	//nInputStatus
	ingPressureControl 		: BOOL;
	ingPositionControl 		: BOOL;
	isValveOpen 			: BOOL;
	isValveNotInitialized 	: BOOL;	
	isValveClosed 			: BOOL;
	isValveFaultState 		: BOOL;
	ingValveInitializing 	: BOOL;
	ingHoldState 			: BOOL;
	isPressureControl:BOOL;
	
	// Vacuum Pump Status
	isPumpFault				: BOOL;
	isPumpWarning			: BOOL;
	isPumpAlarm				: BOOL;
	isFBRunning				: BOOL;
 	isPumpRunning			: BOOL;
	//wSetPoint 			: WORD; //Set Point
	nTValveMode 		: USINT := 0; //Valve Mode
	bPumpOn				: BOOL;
	bPumpReset			: BOOL;	//Input from IQ-PLUS Throttle Valve
	
	wTypedControlValue 	: WORD;
	wOutputSVBytes : outWord; //Word to Byte variable
	nSetType 			: USINT; //1:Pressure Conrol, 2:Position Control
	
	wByteCDG1_PV 			: WORD; //CDG1 Current Pressure, Not Used
	wByteCDG2_PV 			: WORD; //CDG2 Current Pressure
	wByteValvePosition_PV : WORD; //Current Valve Position (0~100%)
	nInputStatusOld : USINT := 9; //Value Change Monitoring, First Temp value
	wByteValvePosition_PV_Monitoring: WORD;
	CDG1_RealValue: REAL;
	nOutputSetType:USINT; //1:Pressure Conrol, 2:Position Control
	CDG_1_Value_RealType: REAL;
END_VAR

VAR CONSTANT
	//Conversion Parameter
	SetPointFactor : REAL := 327.67; //Range 0~7FFFh
	PressureFactor : REAL := 24.576;	//Range 0~6000h
END_VAR

//jhkang_251112
////Model : IQ Plus 
////Pressure Range : 0 ~ 1,000 Torr
//IF GVL_COMMAND_FROM_UI.CMD_THROTTLE_PRESSURE_POSITION_MODE THEN //true: Pressure False:Position
//	GVL_DEVICE_NET_IQ_PLUS.nOutputSetType := 1; // Pressure Control
//ELSE
//	GVL_DEVICE_NET_IQ_PLUS.nOutputSetType := 2; // Position Control
//END_IF

//nSetType := GVL_DEVICE_NET_IQ_PLUS.nOutputSetType;
//nOutputSetType:=nSetType;


//_DIgitalInput();
//_CalData();
//_DigitalOutput();


//nTValveMode := WORD_TO_USINT(GVL_IO.aOutputCmd[2]); //Throttle Valve Mode Setting 0:Normal 1:Close 2:Open 3:Hold 4:Reset

ACTION _CalData:
//jhkang_251112
//// nOutputMode
//// 0 : uses setpoint and setpoint type to control the valve.
//// 1 : Does not use setpoint and setpoint type to operate the valve.
//// 2 : Does not use setpoint and setpoint type to operate the valve.
//// 3 : Holds valve in current position.
//// 4 : Reset the controller.

//GVL_IO.nIQPLUS_SetType 	:= GVL_DEVICE_NET_IQ_PLUS.nOutputSetType;
//GVL_IO.nIQPLUS_Mode 	:= GVL_DEVICE_NET_IQ_PLUS.nOutputMode;
//GVL_DEVICE_NET_IQ_PLUS.nOutputMode := GVL_COMMAND_FROM_UI.CMD_THROTTLE_OUTPUT_MODE;
//GVL_INTERFACE_UI.aMonitoring_PV[E_Morning_Index.E_Morning_TV_Position] := wByteValvePosition_PV/SetPointFactor;

//(* Read from Device Value *)
//// 2USINT to WORD
//wByteCDG1_PV 		:= USINT_TO_WORD_jh(GVL_DEVICE_NET_IQ_PLUS.aInputPressurePV_CDG1);
//wByteCDG2_PV 		:= USINT_TO_WORD_jh(GVL_DEVICE_NET_IQ_PLUS.aInputPressurePV_CDG2);
//wByteValvePosition_PV:= USINT_TO_WORD_jh(GVL_DEVICE_NET_IQ_PLUS.aInputValvePosionPV);
//wByteValvePosition_PV_Monitoring:=REAL_TO_WORD(wByteValvePosition_PV/SetPointFactor);
//GVL_INTERFACE_UI.aMonitoring_PV[12] := wByteValvePosition_PV_Monitoring;




//wControlValue		:= GVL_IO.wIqPlus_CV;

////From IQ Plus
//CDG1_RealValue :=wByteCDG1_PV/PressureFactor; 
//GVL_IO.wIqPlus_CDG1_PV 	:= REAL_TO_WORD(wByteCDG1_PV/PressureFactor);
//GVL_IO.wIqPlus_CDG2_PV:=GVL_IO.wIqPlus_CDG1_PV;

//IF GVL_IO.wIqPlus_CDG1_PV > 1000 OR GVL_IO.wIqPlus_CDG1_PV <=5 THEN
//	GVL_IO.wIqPlus_CDG1_PV:=0;
//	GVL_IO.wIqPlus_CDG2_PV:=0;
//END_IF

//CDG_1_Value_RealType:=wByteCDG1_PV/PressureFactor;


////nSetType //1:Pressure Conrol, 2:Position Control

//IF GVL_DEVICE_NET_IQ_PLUS.nOutputMode = 0 AND nSetType = 1 THEN(*Pressure Mode*)
//	wTypedControlValue := REAL_TO_WORD(wControlValue * SetPointFactor * 0.1); //Pressure Control
//ELSIF GVL_DEVICE_NET_IQ_PLUS.nOutputMode = 0 AND nSetType = 2 THEN (*Position Mode*)
//	wTypedControlValue := REAL_TO_WORD(wControlValue * SetPointFactor); // Position Control
//END_IF

//wOutputSVBytes 		:= WORD_TO_USINT_Bit(wTypedControlValue);
//GVL_DEVICE_NET_IQ_PLUS.aOutputSVBytes[1] 	:= wOutputSVBytes.Lower;
//GVL_DEVICE_NET_IQ_PLUS.aOutputSVBytes[2] 	:= wOutputSVBytes.Upper;

////Valve Status Initailize
//IF GVL_DEVICE_NET_IQ_PLUS.nInputStatus <> nInputStatusOld THEN
//	// Staus Initializing
//	ingPressureControl := FALSE;
//	ingPositionControl := FALSE;
//	isValveOpen := FALSE;
//	isValveNotInitialized := FALSE;	
//	isValveClosed := FALSE;
//	isValveFaultState := FALSE;
//	ingValveInitializing := FALSE;
//	ingHoldState := FALSE;
//	isPressureControl:=FALSE;
//	// Status Update	
//	nInputStatusOld := GVL_DEVICE_NET_IQ_PLUS.nInputStatus;
//END_IF



////Update Valve Status
//CASE GVL_DEVICE_NET_IQ_PLUS.nInputStatus OF
//	0 : ingPressureControl := TRUE; //Pressure Control Performing.
//	1 : ingPositionControl := TRUE; //Position Control Performing.	
//	2 : isValveOpen := TRUE; //Valve Open, Stopped, Not Controlling.
//	3 : isValveNotInitialized := TRUE; //Valve not initialized power on or RESET Command.
//	4 : isValveClosed := TRUE; //Valve Closed, Stopped, Not Controlling.
//	5 : isValveFaultState := TRUE; //Has faulted during valve initialization or operation.
//	6 : ingValveInitializing := TRUE; //Initailizing Process.
//	7 :	isPressureControl:=TRUE;
//	8 : ingHoldState := TRUE; //intermediate position, not at open or close and not controlling pressure.
//END_CASE
END_ACTION

ACTION _DigitalInput:

//jhkang_251112
//(* Command *)

//bPumpOn:= GVL_COMMAND_FROM_UI.CMD_VACUUM_PUMP_ON;
//bPumpReset:=GVL_COMMAND_FROM_UI.CMD_VACUUM_PUMP_RESET;
//(* Read from Power Distribution Pannel *)
//bVacuumPumpCB		:= GVL_IO_GAS_CABINET.DI_02_VacuumPumpELCB;
//bThrottleValveCP 	:= GVL_IO_GAS_CABINET.DI_02_T_VCP;

//(* Read from Vacuum Pump *)
//isPumpFault			:= GVL_IO_REACTOR_CABINET.DI_02_VacuumPumpFail;
//isPumpWarning		:= GVL_IO_REACTOR_CABINET.DI_02_VacuumPumpWarning;
//isPumpAlarm			:= GVL_IO_REACTOR_CABINET.DI_02_VacuumPumpAlarm;
//isPumpRunning		:= GVL_IO_REACTOR_CABINET.DI_02_VacuumPumpFBRunning;
//isFBRunning			:= GVL_IO_REACTOR_CABINET.DI_02_VacuumPumpRunning;


//GVL_IO.isPumpRunning := GVL_IO_REACTOR_CABINET.DI_02_VacuumPumpFBRunning;
END_ACTION

ACTION _DigitalOutput:
//GVL_IO.aDigitalOutputIO[2].2 := bPumpOn; //Pump On
//GVL_IO.aDigitalOutputIO[2].3 := bPumpReset; // Pump Reset

GVL_IO_REACTOR_CABINET.DO_05_VacuumPumpStart_Stop := bPumpOn;
GVL_IO_REACTOR_CABINET.DO_05_VacuumPumpReset := bPumpReset;
END_ACTION

END_PROGRAM

// ---- POUs/P13_LineHeater.TcPOU
PROGRAM P13_LineHeater
VAR
	rTemperatureSV 		: ARRAY[1..8]OF REAL;
	bAutoTuneSV 		: ARRAY[1..8]OF BOOL;

	rTemperaturePV 		: ARRAY[1..8]OF REAL;
	isLineHeater_Run	: ARRAY[1..8]OF BOOL;
	isLineHeater_ATune	: ARRAY[1..8]OF BOOL;
	isLineHeater_Err	: ARRAY[1..8]OF BOOL;

	TimeOnDelay			: TON; //Time delay after Power ON of Thermal Bath
	TimeCycle			: TON;
	nComMode 			: INT; // //1 = PV Req, 2 = STATUS Req, 3 = SV Write, 4 = AutoTune On/Off
	nCount 				: INT;
	rTemperatureTV 		: ARRAY[1..8]OF REAL;
	bAutoTuneTV			: ARRAY[1..8]OF BOOL;

	//for sending variable
	TimeWaitSend		:TON;
	bSendingEnable 		: BOOL:=TRUE; // Check the Sending Stage
	bSetValueMode 		: BOOL;
	fbSend				: SendString;
	sSendString 		: STRING;
	bSendBusy			: BOOL;
	bSendingOK 			: BOOL; //v1
	eSendErrorID		: ComError_t;
	
	// for received variable
	TimeWaitReceive		:TON;
	fbReceive			: ReceiveString;
	sReceivedString		: STRING;
	bStringReceived		: BOOL;
	bReceiveBusy		: BOOL;
	bReceiveError		: BOOL;
	eReceiveErrorID		: ComError_t;
	bReceiveTimeout		: BOOL;
	bReceivedOK 		: BOOL;
	hStrReceivedST		: STRING;
	hStrReceivedPV		: STRING;
	
	nHeaterNumber 		: INT := 1;
	sHeaterNumber 		: STRING := '1';
	sReceivedHeaterNumber : STRING;
	nReceivedHeaterNumber : INT;
	sReceivedAffirmation : STRING;
	sReceivedData 		: STRING;
	nHeaterStrPositionPV : INT:= 11; //Received String Start Position
	nDecimal			:INT;
	nSendStrCounter		:INT := 1;
	bReset : BOOL;
	sTest : STRING;
	nStrPosition : INT;
	nHeaterNumberPV : INT;
	sTemperaturePV : STRING;
	(* Input *)
	bLineHeaterCB		: BOOL;
	bLineHeaterCP		: BYTE;
END_VAR

_DIgitalInput();
TimeOnDelay(IN:= GVL_IO_GAS_CABINET.DI_02_LineHeatersELCB, PT :=T#5S); //Time Delay after a Thermal Bath MC ON

IF TimeOnDelay.Q THEN
	
	_GetSP();
	
	TimeOnDelay(IN:=FALSE);
	FOR nHeaterNumber:= 1 TO 8 DO
		IF (rTemperatureTV[nHeaterNumber] <> rTemperatureSV[nHeaterNumber]) THEN
			rTemperatureTV[nHeaterNumber] := rTemperatureSV[nHeaterNumber];
			
			_SendTemp();
		END_IF
	END_FOR
END_IF


_Update_Data();

ACTION _DigitalInput:
bLineHeaterCB	:= GVL_IO_GAS_CABINET.DI_02_LineHeatersELCB;

bLineHeaterCP.0 	:= GVL_IO_GAS_CABINET.DI_03_LineHeater_1CP;
bLineHeaterCP.1 	:= GVL_IO_GAS_CABINET.DI_03_LineHeater_2CP;
bLineHeaterCP.2 	:= GVL_IO_GAS_CABINET.DI_03_LineHeater_3CP;
bLineHeaterCP.3 	:= GVL_IO_GAS_CABINET.DI_03_LineHeater_4CP;
bLineHeaterCP.4 	:= GVL_IO_GAS_CABINET.DI_03_LineHeater_5CP;
bLineHeaterCP.5 	:= GVL_IO_GAS_CABINET.DI_04_LineHeater_6CP;
bLineHeaterCP.6 	:= GVL_IO_GAS_CABINET.DI_04_LineHeater_7CP;
bLineHeaterCP.7 	:= GVL_IO_GAS_CABINET.DI_04_LineHeater_8CP;
END_ACTION

ACTION _GetSP:
//jhkang_251112
//rTemperatureSV[1] := GVL_IO.aInterlockSet[13];
//rTemperatureSV[2] := GVL_IO.aInterlockSet[14];
//rTemperatureSV[3] := GVL_IO.aInterlockSet[15];
//rTemperatureSV[4] := GVL_IO.aInterlockSet[16];
//rTemperatureSV[5] := GVL_IO.aInterlockSet[17];
//rTemperatureSV[6] := GVL_IO.aInterlockSet[18];
//rTemperatureSV[7] := GVL_IO.aInterlockSet[19];
//rTemperatureSV[8] := GVL_IO.aInterlockSet[20];
END_ACTION

ACTION _SendTemp:
CASE nHeaterNumber OF
	1:
		GVL.fbLineHeater_Manager._SendModbusCommand(sendMessage:=F_Temp_Write_Set_Point(Module_Number:=1,CommandIndex:=16#0
																,Write_Value:=REAL_TO_WORD(rTemperatureSV[nHeaterNumber])));
	2:
		GVL.fbLineHeater_Manager._SendModbusCommand(sendMessage:=F_Temp_Write_Set_Point(Module_Number:=1,CommandIndex:=16#03E8
																,Write_Value:=REAL_TO_WORD(rTemperatureSV[nHeaterNumber])));
	3:
		GVL.fbLineHeater_Manager._SendModbusCommand(sendMessage:=F_Temp_Write_Set_Point(Module_Number:=1,CommandIndex:=16#07D0
																,Write_Value:=REAL_TO_WORD(rTemperatureSV[nHeaterNumber])));
	4:
		GVL.fbLineHeater_Manager._SendModbusCommand(sendMessage:=F_Temp_Write_Set_Point(Module_Number:=1,CommandIndex:=16#0BB8
																,Write_Value:=REAL_TO_WORD(rTemperatureSV[nHeaterNumber])));
																
	(*Change Module Number*)															
	5:
		GVL.fbLineHeater_Manager._SendModbusCommand(sendMessage:=F_Temp_Write_Set_Point(Module_Number:=2,CommandIndex:=16#0
																,Write_Value:=REAL_TO_WORD(rTemperatureSV[nHeaterNumber])));
	6:
		GVL.fbLineHeater_Manager._SendModbusCommand(sendMessage:=F_Temp_Write_Set_Point(Module_Number:=2,CommandIndex:=16#03E8
																,Write_Value:=REAL_TO_WORD(rTemperatureSV[nHeaterNumber])));
	7:
		GVL.fbLineHeater_Manager._SendModbusCommand(sendMessage:=F_Temp_Write_Set_Point(Module_Number:=2,CommandIndex:=16#07D0
																,Write_Value:=REAL_TO_WORD(rTemperatureSV[nHeaterNumber])));
	8:
		GVL.fbLineHeater_Manager._SendModbusCommand(sendMessage:=F_Temp_Write_Set_Point(Module_Number:=2,CommandIndex:=16#0BB8
																,Write_Value:=REAL_TO_WORD(rTemperatureSV[nHeaterNumber])));
END_CASE
END_ACTION

ACTION _Update_Data:
//jhkang_251112

//rTemperaturePV[1] := GVL_Serial.LineHeater_data_1.LINE_HEATER_CH_1_PV_VALUE;
//rTemperaturePV[2] := GVL_Serial.LineHeater_data_1.LINE_HEATER_CH_2_PV_VALUE;
//rTemperaturePV[3] := GVL_Serial.LineHeater_data_1.LINE_HEATER_CH_3_PV_VALUE;
//rTemperaturePV[4] := GVL_Serial.LineHeater_data_1.LINE_HEATER_CH_4_PV_VALUE;

//rTemperaturePV[5] := GVL_Serial.LineHeater_data_2.LINE_HEATER_CH_1_PV_VALUE;
//rTemperaturePV[6] := GVL_Serial.LineHeater_data_2.LINE_HEATER_CH_2_PV_VALUE;
//rTemperaturePV[7] := GVL_Serial.LineHeater_data_2.LINE_HEATER_CH_3_PV_VALUE;
//rTemperaturePV[8] := GVL_Serial.LineHeater_data_2.LINE_HEATER_CH_4_PV_VALUE;

//GVL_IO.aLineHeater_rTemperaturePV := rTemperaturePV;
END_ACTION

END_PROGRAM

// ---- POUs/P14_ThermalBath.TcPOU
PROGRAM P14_ThermalBath
VAR
	rTemperatureSV 		: ARRAY[1..6]OF REAL;

	(* Input from Device *)
	bTempDeviationAlarm	: ARRAY[1..6] OF BOOL;
	bCutOffAlarm		: ARRAY[1..6] OF BOOL;
	
	rTemperature_PV 		: ARRAY[1..6]OF REAL;
	isBath_Err 			: ARRAY[1..6]OF BOOL;
	isBath_TC_Broken 	: ARRAY[1..6]OF BOOL ; 

	//for send variable
	TimeOnDelay	: TON; //Time delay after Power ON of Thermal Bath
	TimeCycle			: TON;
	TimeWaitSend		: TON;
	TimeWaitReceive		: TON;
	bSendingEnable 		: BOOL:=TRUE; // Check the Sending Stage
	bSetValueMode 		: BOOL;
	rTemperatureTV 		: ARRAY[1..6]OF REAL;
	fbSend				: SendString;
	sSendString 		: STRING;
	bSendBusy			: BOOL;
	bSendingOK 			: BOOL;
	eSendErrorID		: ComError_t;

	// for received variable
	fbReceive			: ReceiveString;
	sReceivedString		: STRING;
	bStringReceived		: BOOL;
	bReceiveBusy		: BOOL;
	bReceiveError		: BOOL;
	eReceiveErrorID		: ComError_t;
	bReceiveTimeout		: BOOL;
	bReceivedOK 		: BOOL;
	
	nBathNumber 		: INT := 1;
	sBathNumber 		: STRING := '1';
	sReceivedBathNumber : STRING;
	nReceivedBathNumber : INT;
	sReceivedAffirmation : STRING;
	sReceivedData 		: STRING;
	
	(* Input *)
	bThermalBathCB		: BOOL;
	TonSendTmeOut: TON;
	SendTimeOutCount: DINT;
END_VAR


(* Read from Power Distribution Pannel *)
_DigitalInput();

// make a sending string
TimeCycle(IN := TimeOnDelay.Q, PT := T#1000MS); //Cycle for Serial Communication
IF TimeCycle.Q = TRUE THEN
	TimeCycle(IN := FALSE);
	_01_SendMessage();
END_IF

_02_ReceivedMessage();


TonSendTmeOut(IN:=bSendingEnable = FALSE ,PT:=T#10S);
IF TonSendTmeOut.Q THEN
	SendTimeOutCount := SendTimeOutCount+1;
	
	TonSendTmeOut(IN:=false);
	bSendingEnable:=TRUE;
END_IF

ACTION _01_SendMessage:

// Make a sending string Set value or Request value 
IF bSendingEnable = TRUE THEN
	
	nBathNumber := nBathNumber + 1;
	IF nBathNumber > 4 THEN
		nBathNumber := 1;
	END_IF
	
	bSendingEnable := FALSE;
	bReceivedOK := FALSE;
	bSetValueMode := FALSE;
	
	//Target value(Bath) Set value
	IF (rTemperatureTV[nBathNumber] <> rTemperatureSV[nBathNumber])  THEN
		rTemperatureTV[nBathNumber] := rTemperatureSV[nBathNumber];
		sSendString := Real_To_String_ThermalBath(rTemperatureTV[nBathNumber],nBathNumber); //Send a SetValue=10.0 '$0201WSV100100$03'
		bSetValueMode := TRUE;
	ELSE
		sBathNumber := INT_TO_STRING(nBathNumber);
		sSendString := INSERT('$020RPV1$03',sBathNumber,2); //Request a PV
		bSetValueMode := FALSE;
	END_IF
	
	// Send string	
	fbSend(	SendString:= sSendString,
		TXbuffer:= GVL_Serial.TxBufferTB,
		Busy=> bSendBusy,
		Error=> );
		
	IF fbSend.Error <> COMERROR_NOERROR THEN
		eSendErrorID := fbSend.Error;
		bSendingOK := FALSE;
	ELSE
		eSendErrorID := COMERROR_NOERROR;
		bSendingOK := TRUE;
	END_IF
END_IF
END_ACTION

ACTION _02_ReceivedMessage:
//	Receive string data:
//	The block receives any data strings beginning with a STX ($02) and ending with an ETX ($03) character.
TimeWaitReceive(IN := bSendingOK, PT := T#250MS); //Wait receiving data
IF TimeWaitReceive.Q THEN
	TimeWaitReceive(IN:= FALSE);
	fbReceive(
		Prefix:= '$02',
		Suffix:= '$03',
		Timeout:= T#1S,
		ReceivedString:= sReceivedString,
		RXbuffer:= GVL_Serial.RxBufferTB,
		StringReceived=> bStringReceived,
		Busy=> bReceiveBusy,
		Error=> ,
		RxTimeout=> bReceiveTimeout );
		
	IF bReceiveTimeout THEN
		isBath_Err[nReceivedBathNumber] := TRUE;
		bReceiveTimeout := FALSE;
	END_IF
	
	IF fbReceive.Error <> COMERROR_NOERROR THEN
		eReceiveErrorID := fbReceive.Error;
	END_IF
	
	IF bStringReceived THEN
		bStringReceived :=FALSE;
		bReceivedOK := TRUE;
		bSendingEnable := TRUE;
		sReceivedBathNumber := MID(STR:=sReceivedString, len:=1, pos:=3); //ReceivedString : '$0201$06PV100250$03'
		nReceivedBathNumber := STRING_TO_INT(sReceivedBathNumber);
		sReceivedAffirmation := MID(STR:=sReceivedString, len:=1, pos:=4); //Affirmation
		
		IF bSetValueMode THEN //Write SV Mode
			IF sReceivedAffirmation = '$06' THEN //'$06' ReceivedString : '$0201$06$03'
				isBath_Err[nReceivedBathNumber] := FALSE;
			ELSE
				//isBath_Err[nReceivedBathNumber] := TRUE;
			END_IF
			bSetValueMode := FALSE;
		ELSE //Read PV Mode
			sReceivedData := MID(STR:=sReceivedString, len:=5, pos:=8); //ReceivedString : '$0201$06PV100250$03'
			IF sReceivedData = '' THEN
				isBath_Err[nReceivedBathNumber] := TRUE;
				;
			ELSIF sReceivedData = 'HHHHH' THEN
				rTemperature_PV[nReceivedBathNumber] := -99.0;
				isBath_TC_Broken[nReceivedBathNumber] := TRUE;
				isBath_Err[nReceivedBathNumber] := FALSE;
			ELSE
				rTemperature_PV[nReceivedBathNumber] := (STRING_TO_REAL(sReceivedData))/10;
				isBath_TC_Broken[nReceivedBathNumber] := FALSE;
				isBath_Err[nReceivedBathNumber] := FALSE;
			END_IF
		END_IF
	END_IF
	
	

	bSendingEnable := TRUE;
END_IF
END_ACTION

ACTION _DigitalInput:
//bThermalBathCB := GVL_IO.aDigitalInputIO[5].0;
bThermalBathCB := GVL_IO_GAS_CABINET.DI_02_ThermalBathsELCB;

(* Read from SMC Bath Device Value *)
//TimeOnDelay(IN:= P90_Interlock.bThermalBathMC, PT :=T#1S); //Time Delay after a Thermal Bath MC ON
TimeOnDelay(IN:= GVL_IO_GAS_CABINET.DI_02_ThermalBathsELCB, PT :=T#1S); //Time Delay after a Thermal Bath MC ON

bTempDeviationAlarm[1]	:= GVL_IO_GAS_CABINET.DI_05_ThermalBath_1DeviationAlarm;
bTempDeviationAlarm[2]	:= GVL_IO_GAS_CABINET.DI_05_ThermalBath_2DeviationAlarm;
bTempDeviationAlarm[3]	:= GVL_IO_GAS_CABINET.DI_06_ThermalBath_3DeviationAlarm;
bTempDeviationAlarm[4]	:= GVL_IO_GAS_CABINET.DI_06_ThermalBath_4DeviationAlarm;

bCutOffAlarm[1] := NOT(GVL_IO_GAS_CABINET.DI_05_ThermalBath_1CutOffAlarm); //Normally Contact
bCutOffAlarm[2] := NOT(GVL_IO_GAS_CABINET.DI_05_ThermalBath_2CutOffAlarm); 
bCutOffAlarm[3] := NOT(GVL_IO_GAS_CABINET.DI_06_ThermalBath_3CutOffAlarm); 
bCutOffAlarm[4] := NOT(GVL_IO_GAS_CABINET.DI_06_ThermalBath_4CutOffAlarm);
END_ACTION

END_PROGRAM

// ---- POUs/P15_RotationOperation.TcPOU
PROGRAM P15_RotationOperation
VAR
	rControlValue			: REAL; //rpm
	bStart_Stop				: BOOL := TRUE;
	bAlarmReset				: BOOL; //Motor Driver Alarm

	bRotationCP				: BOOL;
	nConvertedRotation_PV	: REAL; //PV 0~100 rpm

	rConvertedCV			:REAL;
	(* Motor Driver *)
	bBrake_Run				: BOOL;
	(* Rotation Operation Parameter*)
	wRotaion_PV				: WORD;
	isRotationFault			: BOOL; //Motor Driver
	calcRotation: REAL;
END_VAR

VAR CONSTANT
	KL4404MaxValueP		: REAL := 16383; //0~5V, 0~3000
	//Motor Max Rotation RPM 3000rpm, Gear Ratio 20, Belt Ratio 4.5
	ConversionFactor 	: REAL :=491.49;// 491.49 ; //13106 * 20 * 4.5 / 3000
END_VAR

// Oriental Motor Driver : BLHM230K-GFS, 0~4V

_DigitalInput();

calcRotation := (wRotaion_PV / ConversionFactor) * (5.0/3.0);


nConvertedRotation_PV := (calcRotation);

// Interface with other PRGs
GVL_IO.ControlDevice.ROTATION_MOTOR.CURRENT_PV:= nConvertedRotation_PV;
rControlValue := GVL_IO.ControlDevice.ROTATION_MOTOR.SET_CONTROL_VALUE;

//Write to Motor Driver
rConvertedCV := rControlValue * ConversionFactor; // Convert from RPM to control value


IF GVL_INTERFACE_UI.interlock.interlockSetting.aInterlockEnableThreshold[1].enable = TRUE THEN // UI 의 Auto Power ON 기능에 따라서 자동 On . oFF 사용 
	IF (GVL_INTERFACE_UI.aAnalogController[E_aAnalogInputIO_Index.E_PV_susceptorRotation].cvController.input.targetValue > 0) OR (rConvertedCV > 0) THEN // Motor Driver RUN
		bBrake_Run := TRUE;
	ELSIF (GVL_INTERFACE_UI.aAnalogController[E_aAnalogInputIO_Index.E_PV_susceptorRotation].cvController.input.targetValue = 0) AND (rConvertedCV = 0) THEN
		bBrake_Run := FALSE;
	END_IF
ELSE
	bBrake_Run:=FALSE;
END_IF

_DigitalOutput();

ACTION _DigitalInput:
(* Read from Power Distribution Pannel *)
bRotationCP := GVL_IO_GAS_CABINET.DI_02_RotationMotorCP;

//from Device Value
isRotationFault := NOT(GVL_IO_REACTOR_CABINET.DI_02_SusceptorRotationMotorFault);
wRotaion_PV := UINT_TO_WORD(GVL_IO_REACTOR_CABINET.AI_08_R01SusceptorRotationPV);
END_ACTION

ACTION _DigitalOutput:
GVL_IO_REACTOR_CABINET.DO_05_SusceptorRotationFWD := bBrake_Run;
GVL_IO_REACTOR_CABINET.AO_09_R01_SusceptorRotationSV:=REAL_TO_INT(rConvertedCV);
END_ACTION

END_PROGRAM

// ---- POUs/P16_CoverOperation.TcPOU
PROGRAM P16_CoverOperation
VAR
// 	isCoverClosed 	: BOOL;

	bCoverCP	: BOOL;
	bLowerLimit	: BOOL;
	bUpperLimit	: BOOL;
	TimerUpLED 		: TON;
	TimerUpLED_X 	: TON;
	TimerDownLED 	: TON;
	TimerDownLED_X 	: TON;
	TimerDownDelayOff 	: TON;
	(* Input *)
	bUpSwitch	: BOOL;
	bDownSwitch 	: BOOL;
	bClamp_Lock_switch: BOOL;
	bClamp_Release_switch: BOOL;
	(* Output *)
	bUpLED 		: BOOL;
	bDownLED 	: BOOL;
	bOnUpRelay 	: BOOL;
	bOnDownRelay : BOOL;
	bOnClamp_Lock_Relay:BOOL;
	bOnClamp_Release_Relay:BOOL;		
	
	bClampLock: BOOL;
	bClampRelease: BOOL;
END_VAR

_DigitalInput();

TimerDownDelayOff(IN:=bLowerLimit, PT:=T#500MS);

//Cover Open 조건
//공정 중이지 않을것
//Dor Pressure down
//Clamp Releaae
//Susceptor down
//CDG 700 torr 이상
//모든 벨브 ff

// Cover Operation Condition
IF P90_Interlock.bReactorOpenEnable THEN
	(*Cover*)
	IF bClampRelease THEN
		bOnUpRelay := (bDownSwitch = FALSE AND bUpSwitch = TRUE AND bUpperLimit = FALSE );
		bOnDownRelay := (bDownSwitch = TRUE AND bUpSwitch = FALSE AND (bLowerLimit = FALSE OR TimerDownDelayOff.Q = FALSE ));
	ELSE
		bOnUpRelay:=FALSE;
		bOnDownRelay:=FALSE;
	END_IF
	(*clamp*)
	bOnClamp_Lock_Relay:=(bClamp_Lock_switch = TRUE AND bClamp_Release_switch = FALSE);
	bOnClamp_Release_Relay:=(bClamp_Lock_switch = FALSE AND bClamp_Release_switch = TRUE);
ELSE
	(*Cover*)
	bOnUpRelay:=FALSE;
	bOnDownRelay:=FALSE;
	(*clamp*)
	bOnClamp_Lock_Relay:=FALSE;
	bOnClamp_Release_Relay:=FALSE;
END_IF

//LED Blinking
TimerUpLED(IN:=(bOnUpRelay AND TimerUpLED_X.Q = FALSE), PT:=T#500MS);
TimerUpLED_X(IN:=TimerUpLED.Q, PT:=T#300MS);
bUpLED := (TimerUpLED.Q AND bOnUpRelay) OR bUpperLimit;

TimerDownLED(IN:=(bOnDownRelay AND TimerDownLED_X.Q = FALSE), PT:=T#500MS);
TimerDownLED_X(IN:=TimerDownLED.Q, PT:=T#300MS);
bDownLED := (TimerDownLED.Q AND bOnDownRelay) OR bLowerLimit;

_DigitalOutput();

ACTION _DigitalInput:
//(* Read from Device Value *)
//// Cover Operation Switch

bUpSwitch 		:=GVL_IO_REACTOR_CABINET.DI_01_ReactorDoorUpButton;
bDownSwitch 	:=GVL_IO_REACTOR_CABINET.DI_01_ReactorDoorDownButton;
bUpperLimit 	:=GVL_IO_REACTOR_CABINET.DI_02_ReactorDoorUpLimitSensor;
bLowerLimit 	:=GVL_IO_REACTOR_CABINET.DI_03_ReactorDoorDownLimitSensor;
bCoverCP 		:= GVL_IO_GAS_CABINET.DI_02_CoverLiftMotorCP;

bClampLock := GVL_IO_REACTOR_CABINET.DI_03_CylinderAutoSwitch_Closed;
bClampRelease :=GVL_IO_REACTOR_CABINET.DI_03_CylinderAutoSwitch_Opened;

bClamp_Lock_switch:=GVL_IO_REACTOR_CABINET.DI_01_ClampLock;
bClamp_Release_switch:=GVL_IO_REACTOR_CABINET.DI_01_ClampRelease;
END_ACTION

ACTION _DigitalOutput:
//jhkang_251112
//(* Write to Device Value *)
//// Cover Operation Switch Lamp


////Status Output
//GVL_IO.isCoverClosed := bLowerLimit;

//GVL_IO_REACTOR_CABINET.DO_06_ReactorCoverUpButtonLamp := bUpLED;
//GVL_IO_REACTOR_CABINET.DO_06_ReactorCoverDownButtonLamp := bDownLED;

//GVL_IO_REACTOR_CABINET.DO_04_ReactorCoverUpRelay :=bOnUpRelay;
//GVL_IO_REACTOR_CABINET.DO_04_ReactorCoverDownRelay :=bOnDownRelay;

//GVL_IO_REACTOR_CABINET.DO_06_ClampLockButtonLamp := GVL_IO_REACTOR_CABINET.DI_03_CylinderAutoSwitch_Closed;
//GVL_IO_REACTOR_CABINET.DO_06_ClampReleaseButtonLamp := GVL_IO_REACTOR_CABINET.DI_03_CylinderAutoSwitch_Opened;

//GVL_IO_REACTOR_CABINET.DO_05_ClampLock := bOnClamp_Lock_Relay;
//GVL_IO_REACTOR_CABINET.DO_05_ClampRelease := bOnClamp_Release_Relay;
END_ACTION

END_PROGRAM

// ---- POUs/P90_Interlock.TcPOU
PROGRAM P90_Interlock
VAR
	bRecipeRunning 		: BOOL;
	RecipeStopped 		: BOOL;
	ManualOperation 	: BOOL;
	bInductionHeaterMC	: BOOL;
	bThermalBathMC		: BOOL;
	bVacuumPumpMC 		: BOOL;
	bLineHeaterMC 		: BOOL; 

	bRecipeStartAvailable	: BOOL;
	bReactorOpenEnable		: BOOL;
	bHeaterOnEnable			: BOOL;
	bPumpOnEnable			: BOOL;
	
	bDorOnEnable			: BOOL;
	bDorOffEnable			: BOOL;
	bOpenEnableTemp			: BOOL;
	bOpenEnablePress		: BOOL;	
	
	bPowerResetSwitch		: BOOL;
	bMainPowerMonitor		: BOOL;

	AlarmTrig				: BOOL;
	WarningTrig				: BOOL;
	bMaintKey				: BOOL;
	bGasStateProcess		: BOOL; // True가 모든 벨브가 닫힌 상태
	bGasStateSource			: BOOL;// True가 모든 벨브가 닫힌 상태
	bGasStateVent			: BOOL;// True가 모든 벨브가 닫힌 상태

	bPowerResetLED			: BOOL;
	bUPSMode				: BOOL;
	tAlarmDelay_A			: TIME; //아날로그 디바이스 지연시간
	tAlarmDelay_D			: TIME; //디지털 디바이스 지연시간
	
	fbDeviationCheck		:ARRAY[1..29] OF FB_DeviationCheck;
	wDeviceAlarmEnable		: DWORD;
	wDeviceWarningEnable	: DWORD;
	bDeviationAlarm			: BOOL;
	bDeviationWarning		: BOOL;
	wDeviationAlarm			: DWORD;
	wDeviationWarning		: DWORD;

	wLimitAlarmEnable		: DWORD;
	wLimitWarningEnable		: DWORD;
	bLimitAlarm				: BOOL;
	bLimitWarning			: BOOL;
	wLimitAlarm				: DWORD;
	wLimitWarning			: DWORD;
	
	wAlarmEnable			: DWORD;
	wWarningEnable			: DWORD;

	bFaultAlarm				: BOOL;
	bFaultWarning			: BOOL;
	wAlarm					: DWORD;
	wWarning				: DWORD;
		
	bAlarmEnable			: BOOL;
	bWarningEnable			: BOOL;
	bDeviceCurrentAlarmState	: BOOL;
	bDeviceCurrentWarningState 	: BOOL;
	fDeviceCurrentValue			: REAL;
	fDeviceAlarmTreshold		: REAL;
	fDeviceWarningTreshold		: REAL;
	
	i	: UINT;
	j 	: INT;

//jhkang_251112
//	fReactorIndexToAnalogControllerIndex : F_ReactorIndexToAnalogControllerIndex;

END_VAR

//jhkang_251112 인터락은 재 확인 필요

//(* Read from Device*)
//_DigitalInput();

//bGasStateProcess := F_StateValve_Process();  // True 가  Close 상태
//bGasStateSource := F_StateValve_Process_Source(); // Process gas safety / Source Carier Gas
//bGasStateVent := F_State_All_Valve_Vent();//벤트 가능 조건

//GVL_IO.aInterlock[1].10 := bRecipeStartAvailable;
//GVL_IO.aInterlock[1].11 := bReactorOpenEnable;
//GVL_IO.aInterlock[1].12 := bPumpOnEnable;
////알람 지연 시간 변환
//tAlarmDelay_A := REAL_TO_TIME(GVL_IO.aInterlockSet[3]*1000); // UI Setting Analog Delay Time Value(Miliseconde)
//tAlarmDelay_D := REAL_TO_TIME(GVL_IO.aInterlockSet[4]*1000); // UI Setting Analog Delay Time Value(Miliseconde)

//IF bMaintKey THEN //bMaintKey 변경
//	GVL_IO.nCaseSignalTower	:= 4; //Signal Tower Blue - Maintenance
//	GVL_COMMAND_FROM_UI.CMD_HEATER_MAIN_MC_ON := GVL_IO.aOutputCmd[1].0;
//	GVL_COMMAND_FROM_UI.CMD_THERMAL_BACH_MC_ON:=GVL_IO.aOutputCmd[1].1;
//	GVL_COMMAND_FROM_UI.CMD_VACUUM_PUMP_MC_ON:=GVL_IO.aOutputCmd[1].2;
//	GVL_COMMAND_FROM_UI.CMD_LINE_HEATER_MC_ON:=GVL_IO.aOutputCmd[1].3;
//ELSE
//	_100_Alarm_Pressure_Low();
//	_101_Alarm_MFC_EPC();
//	_102_Alarm_Reactor_Temp_Pre_Rotation();
//	_103_Alarm_Reactor_OverPre_Temp();
//	_104_Alarm_Utility();	
//	_105_Alarm_Utility_Parts();
//	_Button_Reset_Warning();
//END_IF

//_01_Enable_RunRecipe();
//_02_Enable_Reactor_Open_Dor_Off();
//_03_Enable_DOR_ON();
//_04_Enable_Heater_ON();
//_05_Enable_OpenPressure();
//_06_Enable_OpenTemp();
//_07_Enable_PumpTurnOn();


//(* Out to Device*)
//GVL_IO.aDigitalOutputIO[3].7 := bPowerResetLED;
//GVL_IO.aDigitalOutputIO[2].4 := bUPSMode;

ACTION _01_Enable_RunRecipe:
// bRecipeStartAvailable := //레시피 가능한 상태이면 TRUE
// 	(AlarmTrig = FALSE) AND
// 	(WarningTrig = FALSE) AND
// 	(bMaintKey = FALSE ) AND
//	(GVL_IO.bDORState = TRUE) AND //DOR ON 상태
//// 	(RCP.userState <> 10) AND //Not Recipe Run State
// 	(GVL_IO_REACTOR_CABINET.DI_03_ReactorDoorDownLimitSensor = TRUE ) AND //Cover Lower Limt
// 	(bGasStateProcess = TRUE ) AND //Safety Process Gas : TRUE
// 	(bGasStateSource = TRUE ) AND //Safety Source Gas : TRUE
// 	(bGasStateVent = TRUE ) AND  //safety Vent Vlave : true
//	(GVL_IO_VALVE.DO_00_V21PumpByPass = TRUE) AND
// 	GVL_IO.nE3508_nInputManAutoBytes.0 = FALSE AND //Temperature Controller Auto : false
//	GVL_DEVICE_NET_IQ_PLUS.nOutputSetType = 1 AND
//	GVL_IO_REACTOR_CABINET.DI_03_CylinderAutoSwitch_Closed = TRUE ; 
	 
////jhkang 임시  on
//bRecipeStartAvailable:=TRUE; 


//GVL_IO.UI_INTERLOCK_CHECK_RECIPE_ENABLE.0:=(AlarmTrig = FALSE); //알람 상태 아닐것
//GVL_IO.UI_INTERLOCK_CHECK_RECIPE_ENABLE.1:=(WarningTrig = FALSE); // 어닝 상태 사닐것
//GVL_IO.UI_INTERLOCK_CHECK_RECIPE_ENABLE.2:=(bMaintKey = FALSE); // 메인트키 
//GVL_IO.UI_INTERLOCK_CHECK_RECIPE_ENABLE.3:=(GVL_IO.bDORState = TRUE ); //DOR ON
////GVL_IO.UI_INTERLOCK_CHECK_RECIPE_ENABLE.4:=RCP.userState <> 10; // Recipe Not Running
//GVL_IO.UI_INTERLOCK_CHECK_RECIPE_ENABLE.4:=GVL_IO_REACTOR_CABINET.DI_03_ReactorDoorDownLimitSensor = TRUE;  //Chamber Close
//GVL_IO.UI_INTERLOCK_CHECK_RECIPE_ENABLE.5:=bGasStateProcess;  // Gas Valve Close
//GVL_IO.UI_INTERLOCK_CHECK_RECIPE_ENABLE.6:=bGasStateSource; // Source Valve Close
//GVL_IO.UI_INTERLOCK_CHECK_RECIPE_ENABLE.7:=bGasStateVent;//Vent Valve Close
//GVL_IO.UI_INTERLOCK_CHECK_RECIPE_ENABLE.8:=(GVL_IO_VALVE.DO_00_V21PumpByPass = TRUE);  // Valve 21 open
//GVL_IO.UI_INTERLOCK_CHECK_RECIPE_ENABLE.9:=GVL_IO.nE3508_nInputManAutoBytes.0 = FALSE;  // Temp Auto Mode
//GVL_IO.UI_INTERLOCK_CHECK_RECIPE_ENABLE.10:=GVL_DEVICE_NET_IQ_PLUS.nOutputSetType = 1;  // Temp Auto Mode
//GVL_IO.UI_INTERLOCK_CHECK_RECIPE_ENABLE.11:=GVL_IO_REACTOR_CABINET.DI_03_CylinderAutoSwitch_Closed = TRUE;  // Chamber Clamp Close
END_ACTION

ACTION _02_Enable_Reactor_Open_Dor_Off:
//// DOR Off Conditions
////jhkang (GVL_IO.aInterlockEnable[1].3 = FALSE ) AND //Can Open Temperature Check
////왜 UI 에서 설정되는 Can OPen Temp / Pressure 를 확인 하는지 ? 
 
//bReactorOpenEnable :=
//	(AlarmTrig = FALSE) AND
//	bOpenEnableTemp = TRUE AND
//	bOpenEnablePress= TRUE AND
//	(GVL_IO.bDORState = FALSE) AND  // DOR oFF
//	(RCP.userState <> 10) AND //Not Recipe Run State
//	(bGasStateProcess = TRUE ) AND //Safety Process Gas : TRUE
// 	(bGasStateSource = TRUE ) AND //Safety Source Gas : TRUE
// 	(bGasStateVent = TRUE ) AND  //safety Vent Vlave : true
//	(GVL_IO.aInterlockEnable[1].3 = TRUE ) AND //Can Open Temperature Check
//	(GVL_IO.aInterlockEnable[1].4 = TRUE ); //Can Open Pressure Check

//bDorOffEnable:=
//	(AlarmTrig = FALSE) AND
//	bOpenEnableTemp = TRUE AND
//	bOpenEnablePress= TRUE AND
////	(GVL_IO.bDORState = FALSE) AND  // DOR oFF
//	(RCP.userState <> 10) AND //Not Recipe Run State
//	(bGasStateProcess = TRUE ) AND //Safety Process Gas : TRUE
// 	(bGasStateSource = TRUE ) AND //Safety Source Gas : TRUE
// 	(bGasStateVent = TRUE ) AND  //safety Vent Vlave : true
//	(GVL_IO.aInterlockEnable[1].3 = TRUE ) AND //Can Open Temperature Check
//	(GVL_IO.aInterlockEnable[1].4 = TRUE ); //Can Open Pressure Check


	
//GVL_IO.UI_INTERLOCK_CHECK_OPEN_REACTOR.0 := (AlarmTrig = FALSE);  //알람 상태 아닐것
//GVL_IO.UI_INTERLOCK_CHECK_OPEN_REACTOR.1 := bOpenEnableTemp;  // Open Temp
//GVL_IO.UI_INTERLOCK_CHECK_OPEN_REACTOR.2 := bOpenEnablePress;// Open Pressure
//GVL_IO.UI_INTERLOCK_CHECK_OPEN_REACTOR.3 := GVL_IO.bDORState = FALSE; // Dor False
//GVL_IO.UI_INTERLOCK_CHECK_OPEN_REACTOR.4 := RCP.userState <> 10; // Recipe Not Running
//GVL_IO.UI_INTERLOCK_CHECK_OPEN_REACTOR.5 := bGasStateProcess;// Gas Valve Close
//GVL_IO.UI_INTERLOCK_CHECK_OPEN_REACTOR.6 := bGasStateSource;// Source Valve Close
//GVL_IO.UI_INTERLOCK_CHECK_OPEN_REACTOR.7 := bGasStateVent;// Vent Valve Close
//GVL_IO.UI_INTERLOCK_CHECK_OPEN_REACTOR.8 := GVL_IO.aInterlockEnable[1].3 = TRUE; // UI 에서 Temp Interlock 설정
//GVL_IO.UI_INTERLOCK_CHECK_OPEN_REACTOR.9 := GVL_IO.aInterlockEnable[1].4 = TRUE;// UI 에서 Pressure Interlock 설정
END_ACTION

ACTION _03_Enable_DOR_ON:
////jhkang Dor ON 조건 다시 확인 필요
//bDorOnEnable :=	(AlarmTrig = FALSE ) AND 
//				GVL_IO.isCoverClosed AND 
////				GVL_IO.bDorState = FALSE AND
//				(RCP.userState <> 10) AND //Not Recipe Run State 
//				GVL_IO.isPumpRunning;

//GVL_IO.bDorOnEnable := bDorOnEnable;
END_ACTION

ACTION _04_Enable_Heater_ON:
//bHeaterOnEnable := (AlarmTrig = FALSE ) AND 
//				(GVL_IO_REACTOR_CABINET.DI_03_ReactorDoorDownLimitSensor = TRUE ) AND //Cover Lower Limt;
//				GVL_IO.bDorState = TRUE AND
//				(RCP.userState <> 10); //Not Recipe Run State
END_ACTION

ACTION _05_Enable_OpenPressure:
//IF  GVL_IO.wIqPlus_CDG1_PV > GVL_IO.aInterlockSet[10] THEN  //Can Open Reactor Pressure
//	bOpenEnablePress := TRUE;
//ELSE
//	bOpenEnablePress := FALSE;
//END_IF
END_ACTION

ACTION _06_Enable_OpenTemp:
////jhkang Can Open Temp 가 3508 온도 맞는지?
//IF  P11_E3508.wE3508_PV < GVL_IO.aInterlockSet[9] THEN  // Can Open Temp
//	bOpenEnableTemp := TRUE;
//ELSE
//	bOpenEnableTemp := FALSE;
//END_IF
END_ACTION

ACTION _07_Enable_PumpTurnOn:
//bPumpOnEnable :=  // Pump ON 
//	(AlarmTrig = FALSE) AND
//	(GVL_IO_REACTOR_CABINET.DI_03_ReactorDoorDownLimitSensor = TRUE );
END_ACTION

ACTION _100_Alarm_Pressure_Low:
////Gas Pressure Alarm N2, H2, H2S, H2Se
//FOR i := 1 TO 4 DO
//	wLimitAlarmEnable := SHR(GVL_IO.aInterlockEnable[4], (i-1)); 
//	wLimitWarningEnable := SHR(GVL_IO.aInterlockEnable[5], (i-1));
//	GVL_SEQUENCE.fbSensorLimitCheck[i](
//		bAlarmEnable := wLimitAlarmEnable.0,  // Enable 
//		bWarningEnable := wLimitWarningEnable.0,
//		fCurrentValue := GVL_INTERFACE_UI.aMonitoring_PV[(i+3)], // 현재 값 
//		fAlarmTreshold := GVL_IO.aInterlockSet[5],
//		fWarningTreshold := GVL_IO.aInterlockSet[6],
//		tAlarmDelay := tAlarmDelay_D,
//		bLimitAlarm => bLimitAlarm, //알람 출력
//		bLimitWarning => bLimitWarning //주의(Warning) 출력
//		);	


//	IF bLimitAlarm THEN		
//		GVL_IO.aInterlock[1].0 := TRUE; //Alarm Trig
//		GVL_IO.nCaseSignalTower := 1; // Signal Tower RED - Alarm
//		//팝업 표시
//		wLimitAlarm := ROR(GVL_IO.aInterlock[2], (i-1));
//		wLimitAlarm.0 := TRUE;
//		GVL_IO.aInterlock[2] := ROL(wLimitAlarm, (i-1));
//		//대시보드 표시
//		wLimitAlarm := ROR(GVL_IO.aInterlock[1], (i*2));
//		wLimitAlarm.0 := TRUE;
//		GVL_IO.aInterlock[1] := ROL(wLimitAlarm, (i*2));
//	ELSE
//		//팝업 표시
//		wLimitAlarm := ROR(GVL_IO.aInterlock[2], (i-1));
//		wLimitAlarm.0 := FALSE;
//		GVL_IO.aInterlock[2] := ROL(wLimitAlarm, (i-1));
//		//대시보드 표시
//		wLimitAlarm := ROR(GVL_IO.aInterlock[1], (i*2));
//		wLimitAlarm.0 := FALSE;
//		GVL_IO.aInterlock[1] := ROL(wLimitAlarm, (i*2));
//	END_IF
	
//	IF bLimitWarning THEN		
//		GVL_IO.aInterlock[1].1 := TRUE; //Warning Trig
//		GVL_IO.nCaseSignalTower := 2; // Signal Tower YELLOW - Warning
//		//팝업 표시
//		wLimitWarning := ROR(GVL_IO.aInterlock[4], (i-1));
//		wLimitWarning.0 := TRUE;
//		GVL_IO.aInterlock[4] := ROL(wLimitWarning, (i-1));
//		//대시보드 표시
//		wLimitWarning := ROR(GVL_IO.aInterlock[1], (i*2)+1);
//		wLimitWarning.0 := TRUE;
//		GVL_IO.aInterlock[1] := ROL(wLimitWarning, (i*2)+1);
//	ELSE
//		//팝업 표시
//		wLimitWarning := ROR(GVL_IO.aInterlock[4], (i-1));
//		wLimitWarning.0 := FALSE;
//		GVL_IO.aInterlock[4] := ROL(wLimitWarning, (i-1));
//		//대시보드 표시
//		wLimitWarning := ROR(GVL_IO.aInterlock[1], (i*2)+1);
//		wLimitWarning.0 := FALSE;
//		GVL_IO.aInterlock[1] := ROL(wLimitWarning, (i*2)+1);
//	END_IF
//END_FOR
END_ACTION

ACTION _101_Alarm_MFC_EPC:
////jhkang MFC ,EPC
//FOR i := 1 TO GVL_CONSTANT.NumFlowController DO
//		wDeviceAlarmEnable := SHR(GVL_IO.aInterlockEnable[2], (i+2)); //오늘쪽 쉬프트 연산
//		wDeviceWarningEnable := SHR(GVL_IO.aInterlockEnable[3], (i+2));
		
//		GVL_SEQUENCE.fbDeviationCheck[i](
//			bAlarmEnable := wDeviceAlarmEnable.0,
//			bWarningEnable := wDeviceWarningEnable.0,
//			fCurrentValue := GVL_INTERFACE_UI.aAnalogController[i].pv,
//			fControlValue := LREAL_TO_REAL(GVL_INTERFACE_UI.aAnalogController[i].cvController.rControlValue),
//			fMaxValue := GVL_CONSTANT.AnalogControllerOutputVoltage,
//			fAlarmTreshold := GVL_IO.aInterlockSet[1],
//			fWarningTreshold := GVL_IO.aInterlockSet[2],
//			tAlarmDelay := tAlarmDelay_A,
//			bDeviationAlarm => bDeviationAlarm, //알람 출력
//			bDeviationWarning => bDeviationWarning // 주의(Warning) 출력
//			);
			
//		IF bDeviationAlarm THEN
//			GVL_IO.aInterlock[1].0 := TRUE; //Alarm Trig
//			GVL_IO.nCaseSignalTower := 1; // Signal Tower RED - Alarm
//			wDeviationAlarm := ROR(GVL_IO.aInterlock[3], (i+2));
//			wDeviationAlarm.0 := TRUE;
//			GVL_IO.aInterlock[3] := ROL(wDeviationAlarm, (i+2));
//		ELSE
//			wDeviationAlarm := ROR(GVL_IO.aInterlock[3], (i+2));
//			wDeviationAlarm.0 := FALSE;
//			GVL_IO.aInterlock[3] := ROL(wDeviationAlarm, (i+2));	
//		END_IF
		
//		IF bDeviationWarning THEN
//			GVL_IO.aInterlock[1].1 := TRUE; // Warning Trig
//			GVL_IO.nCaseSignalTower := 2; // Signal Tower Yellow - Warning
//			wDeviationWarning := ROR(GVL_IO.aInterlock[5], (i+2));
//			wDeviationWarning.0 := TRUE;
//			GVL_IO.aInterlock[5] := ROL(wDeviationWarning, (i+2));
//		ELSE
//			wDeviationWarning := ROR(GVL_IO.aInterlock[5], (i+2));
//			wDeviationWarning.0 := FALSE;
//			GVL_IO.aInterlock[5] := ROL(wDeviationWarning, (i+2));
//		END_IF
//	END_FOR
END_ACTION

ACTION _102_Alarm_Reactor_Temp_Pre_Rotation:
////jhkang Reactor Temp , Pressure ,Rotation

//FOR i := 1 TO GVL_CONSTANT.NumReactor DO
//		wDeviceAlarmEnable := SHR(GVL_IO.aInterlockEnable[2], (i-1)); //오늘쪽 쉬프트 연산
//		wDeviceWarningEnable := SHR(GVL_IO.aInterlockEnable[3], (i-1));
		
//		GVL_SEQUENCE.fbDeviationCheck_Reactor[i](
//			bAlarmEnable := wDeviceAlarmEnable.0,
//			bWarningEnable := wDeviceWarningEnable.0,
//			fCurrentValue := GVL_INTERFACE_UI.aAnalogController[fReactorIndexToAnalogControllerIndex(i)].pv,
//			fControlValue := LREAL_TO_REAL(GVL_INTERFACE_UI.aAnalogController[fReactorIndexToAnalogControllerIndex(i)].cvController.rControlValue),
//			fMaxValue := GVL_IO.aReactorMaxValue[i],
//			fAlarmTreshold := GVL_IO.aInterlockSet[1],
//			fWarningTreshold := GVL_IO.aInterlockSet[2],
//			tAlarmDelay := tAlarmDelay_A,
//			bDeviationAlarm => bDeviationAlarm, //알람 출력
//			bDeviationWarning => bDeviationWarning // 주의(Warning) 출력
//			);
			
//		IF bDeviationAlarm THEN
//			GVL_IO.aInterlock[1].0 := TRUE; //Alarm Trig
//			GVL_IO.nCaseSignalTower := 1; // Signal Tower RED - Alarm
//			wDeviationAlarm := ROR(GVL_IO.aInterlock[3], (i-1));
//			wDeviationAlarm.0 := TRUE;
//			GVL_IO.aInterlock[3] := ROL(wDeviationAlarm, (i-1));
//		ELSE
//			wDeviationAlarm := ROR(GVL_IO.aInterlock[3], (i-1));
//			wDeviationAlarm.0 := FALSE;
//			GVL_IO.aInterlock[3] := ROL(wDeviationAlarm, (i-1));	
//		END_IF
		
//		IF bDeviationWarning THEN
//			GVL_IO.aInterlock[1].1 := TRUE; // Warning Trig
//			GVL_IO.nCaseSignalTower := 2; // Signal Tower Yellow - Warning
//			wDeviationWarning := ROR(GVL_IO.aInterlock[5], (i-1));
//			wDeviationWarning.0 := TRUE;
//			GVL_IO.aInterlock[5] := ROL(wDeviationWarning, (i-1));
//		ELSE
//			wDeviationWarning := ROR(GVL_IO.aInterlock[5], (i-1));
//			wDeviationWarning.0 := FALSE;
//			GVL_IO.aInterlock[5] := ROL(wDeviationWarning, (i-1));
//		END_IF
//	END_FOR
END_ACTION

ACTION _103_Alarm_Reactor_OverPre_Temp:

////Over Temp Over Pressure
//FOR i := 1 TO 2 DO
//	CASE i OF
		
//		1: //Susceptor Over Temperature
//			bAlarmEnable := GVL_IO.aInterlockEnable[4].4;
//			bWarningEnable := GVL_IO.aInterlockEnable[5].4;
//			fDeviceCurrentValue := P11_E3508.wE3508_PV;
//			fDeviceAlarmTreshold := GVL_IO.aInterlockSet[7];
//			fDeviceWarningTreshold := (GVL_IO.aInterlockSet[7] * 0.9); // 90% 이상 warning 
		
//		2: //Reactor Over Pressure Alarm
//			bAlarmEnable := GVL_IO.aInterlockEnable[4].5;
//			bWarningEnable := GVL_IO.aInterlockEnable[5].5;
//			fDeviceCurrentValue := GVL_IO.wIqPlus_CDG1_PV;
//			fDeviceAlarmTreshold := GVL_IO.aInterlockSet[8];
//			fDeviceWarningTreshold := (GVL_IO.aInterlockSet[8] * 0.9); //
			
//	END_CASE
	
//	GVL_SEQUENCE.fbSensorOverLimitCheck[i](
//		bAlarmEnable	 := bAlarmEnable,  // Enable 
//		bWarningEnable	 := bWarningEnable,
//		fCurrentValue  := fDeviceCurrentValue, // 현재 값 
//		fAlarmTreshold	 := fDeviceAlarmTreshold,
//		fWarningTreshold  := fDeviceWarningTreshold,
//		tAlarmDelay := tAlarmDelay_D,
//		bAlarm => bLimitAlarm, //알람 출력
//		bWarning => bLimitWarning //주의(Warning) 출력
//		);
	
//		IF bLimitAlarm THEN
//			GVL_IO.aInterlock[1].0 := TRUE; //Alarm Trig
//			GVL_IO.nCaseSignalTower := 1; // Signal Tower RED - Alarm
//			wDeviationAlarm := ROR(GVL_IO.aInterlock[2], (i+3));
//			wDeviationAlarm.0 := TRUE;
//			GVL_IO.aInterlock[2] := ROL(wDeviationAlarm, (i+3));
//		ELSE
//			wDeviationAlarm := ROR(GVL_IO.aInterlock[2], (i+3));
//			wDeviationAlarm.0 := FALSE;
//			GVL_IO.aInterlock[2] := ROL(wDeviationAlarm, (i+3));	
//		END_IF
		
//		IF bLimitWarning THEN
//			GVL_IO.aInterlock[1].1 := TRUE; // Warning Trig
//			GVL_IO.nCaseSignalTower := 2; // Signal Tower Yellow - Warning
//			wDeviationWarning := ROR(GVL_IO.aInterlock[4], (i+3));
//			wDeviationWarning.0 := TRUE;
//			GVL_IO.aInterlock[4] := ROL(wDeviationWarning, (i+3));
//		ELSE
//			wDeviationWarning := ROR(GVL_IO.aInterlock[4], (i+3));
//			wDeviationWarning.0 := FALSE;
//			GVL_IO.aInterlock[4] := ROL(wDeviationWarning, (i+3));
//		END_IF
//END_FOR
END_ACTION

ACTION _104_Alarm_Utility:
//	//Device Fault Check - Pneumatic, Heater, Pump, Motor, GC Door, RC Door
//	FOR i := 1 TO 7 DO
//		CASE i OF
//			1: //CDA Alarm Switch (Pneumatic)
//				bAlarmEnable := GVL_IO.aInterlockEnable[4].6;
//				bWarningEnable := GVL_IO.aInterlockEnable[5].6;
//				bDeviceCurrentAlarmState := NOT GVL_IO.aInputState[1].3;
//				bDeviceCurrentWarningState := NOT GVL_IO.aInputState[1].3;
				
//			2: //Cooling Water Switch
//				bAlarmEnable := GVL_IO.aInterlockEnable[4].7;
//				bWarningEnable := GVL_IO.aInterlockEnable[5].7;
//				bDeviceCurrentAlarmState := NOT GVL_IO.aInputState[1].4;
//				bDeviceCurrentWarningState := NOT GVL_IO.aInputState[1].4;
				
//			3: //Rotatin Motor Fault
//				bAlarmEnable := GVL_IO.aInterlockEnable[4].8;
//				bWarningEnable := GVL_IO.aInterlockEnable[5].8;
//				bDeviceCurrentAlarmState :=  GVL_IO.aInputState[1].7;
//				bDeviceCurrentWarningState :=  GVL_IO.aInputState[1].7;
				
//			4: //Vacuum Pump Fault
//				bAlarmEnable := GVL_IO.aInterlockEnable[4].9;
//				bWarningEnable := GVL_IO.aInterlockEnable[5].9;
//				bDeviceCurrentAlarmState := NOT GVL_IO.aInputState[1].10;
//				bDeviceCurrentWarningState := NOT GVL_IO.aInputState[1].9;
				
//			5: //Gas Cabinet Door Open
//				bAlarmEnable := GVL_IO.aInterlockEnable[4].10;
//				bWarningEnable := GVL_IO.aInterlockEnable[5].10;
//				bDeviceCurrentAlarmState := NOT GVL_IO.aInputState[1].15;
//				bDeviceCurrentWarningState := NOT GVL_IO.aInputState[1].15;
//			6: //Reactor Cabinet Door Open
//				bAlarmEnable := GVL_IO.aInterlockEnable[4].11;
//				bWarningEnable := GVL_IO.aInterlockEnable[5].11;
//				bDeviceCurrentAlarmState := NOT GVL_IO.aInputState[1].13;
//				bDeviceCurrentWarningState := NOT GVL_IO.aInputState[1].13;
				
//			7: //DOR Fault
//				bAlarmEnable := GVL_IO.aInterlockEnable[4].12;
//				bWarningEnable := GVL_IO.aInterlockEnable[5].12;
				
//				IF (GVL_IO.nDorOperationError = 1) THEN
//					bDeviceCurrentAlarmState := TRUE;
//				ELSE
//					bDeviceCurrentAlarmState := FALSE;
//				END_IF
//				IF (GVL_IO.nDorOperationError = 2) OR (GVL_IO.nDorOperationError = 3) THEN
//					bDeviceCurrentWarningState := TRUE;
//					bDeviceCurrentAlarmState:=TRUE;
//				ELSE
//					bDeviceCurrentWarningState := FALSE;
//					bDeviceCurrentAlarmState:=FALSE;
//				END_IF
//		END_CASE

//		GVL_SEQUENCE.fbFaultCheck[i](
//			bAlarmEnable := bAlarmEnable,
//			bWarningEnable := bWarningEnable,
//			bCurrentAlarmState := bDeviceCurrentAlarmState,
//			bCurrentWarningState := bDeviceCurrentWarningState,
//			tAlarmDelay := tAlarmDelay_D,
//			bAlarm => bFaultAlarm,
//			bWarning => bFaultWarning
//			);
			
//		IF bFaultAlarm THEN
//			GVL_IO.aInterlock[1].0 := TRUE; //Alarm Trig
//			GVL_IO.nCaseSignalTower := 1; // Signal Tower RED - Alarm
//			//팝업 표시
//			wAlarm := ROR(GVL_IO.aInterlock[2], (i+5));
//			wAlarm.0 := TRUE;
//			GVL_IO.aInterlock[2] := ROL(wAlarm, (i+5));
//		END_IF
//		IF bFaultWarning THEN
//			GVL_IO.aInterlock[1].1 := TRUE; //Warning Trig
//			GVL_IO.nCaseSignalTower := 2; // Signal Tower YELLOW - Warning
//			//팝업 표시
//			wAlarm := ROR(GVL_IO.aInterlock[4], (i+5));
//			wAlarm.0 := TRUE;
//			GVL_IO.aInterlock[4] := ROL(wAlarm, (i+5));
//		END_IF
//	END_FOR
END_ACTION

ACTION _105_Alarm_Utility_Parts:
////SMPS,Circuit Power , Gas Detector ,
//	FOR i := 1 TO 4 DO
//		CASE i OF
//			1: //SMPS
//				bAlarmEnable := GVL_IO.aInterlockEnable[4].13;
//				bDeviceCurrentAlarmState := GVL_IO.aInputState[2].5 OR 
//											GVL_IO.aInputState[2].6 OR 
//											GVL_IO.aInputState[2].7 OR 
//											GVL_IO.aInputState[2].8;
//			2: //Circuit Power
//				bAlarmEnable := GVL_IO.aInterlockEnable[4].14;
//				bDeviceCurrentAlarmState := GVL_IO.aInputState[2].13 = FALSE  OR  
//											GVL_IO.aInputState[2].14 = FALSE  OR
//											GVL_IO.aInputState[2].15 = FALSE  OR
//											GVL_IO.aInputState[3].0 = FALSE  OR 
//											GVL_IO.aInputState[3].1 = FALSE  OR
//											GVL_IO.aInputState[3].2  = FALSE;
//				//bDeviceCurrentAlarmState 가 true 면 알람 상태 
				
//		//GVL_IO.aInputState[2].13:= GVL_IO_GAS_CABINET.DI_02_RotationMotorCP;
//		//GVL_IO.aInputState[2].14:= GVL_IO_GAS_CABINET.DI_02_CoverLiftMotorCP;
//		//GVL_IO.aInputState[2].15:= GVL_IO_GAS_CABINET.DI_02_T_VCP;
		
//		//GVL_IO.aInputState[3].0:= GVL_IO_GAS_CABINET.DI_03_GasDetectorCP;
//		//GVL_IO.aInputState[3].1:= GVL_IO_GAS_CABINET.DI_03_CabinetLampsCP;
//		//GVL_IO.aInputState[3].2:= GVL_IO_GAS_CABINET.DI_03_MFCPowerCP;

//			3: //Gas Detector
//				bAlarmEnable := GVL_IO.aInterlockEnable[4].15;
//				bDeviceCurrentAlarmState := GVL_IO.aInputState[3].11 AND GVL_IO.aInputState[3].12 AND GVL_IO.aInputState[3].13 AND GVL_IO.aInputState[3].14;
				

//		//GVL_IO.aInputState[3].11:= GVL_IO_GAS_CABINET.DI_04_GasDetectorH2;
//		//GVL_IO.aInputState[3].12:= GVL_IO_GAS_CABINET.DI_04_GasDetectorH2S;
//		//GVL_IO.aInputState[3].13:= GVL_IO_GAS_CABINET.DI_04_GasDetectorH2Se;
//		//GVL_IO.aInputState[3].14:= GVL_IO_GAS_CABINET.DI_04_FireSensor;
//			4: // External Alarm
//				bAlarmEnable := GVL_IO.aInterlockEnable[4].16;
//				bDeviceCurrentAlarmState := GVL_IO.aInputState[3].14 AND GVL_IO.aInputState[3].15 AND GVL_IO.aInputState[4].0 AND GVL_IO.aInputState[4].1 AND GVL_IO.aInputState[4].2
//														AND GVL_IO.aInputState[4].3 AND GVL_IO.aInputState[4].4;
				
						
//		//GVL_IO.aInputState[3].14:= GVL_IO_GAS_CABINET.DI_04_FireSensor;
//		//GVL_IO.aInputState[3].15 := GVL_IO_GAS_CABINET.DI_04_ExternalScrubberFault;
//		//GVL_IO.aInputState[4].0 := GVL_IO_GAS_CABINET.DI_05_ExternalH2GasCabinetFault;
//		//GVL_IO.aInputState[4].1 := GVL_IO_GAS_CABINET.DI_05_ExternalH2SGasCabinetFault;
//		//GVL_IO.aInputState[4].2 := GVL_IO_GAS_CABINET.DI_05_ExternalH2SeGasCabinetFault;
//		//GVL_IO.aInputState[4].3 := GVL_IO_GAS_CABINET.DI_05_ExternalUserInputAlarm;

//		END_CASE

//		GVL_SEQUENCE.fbFaultCheck_Utility_CP[i](
//			bAlarmEnable := bAlarmEnable,
//			bWarningEnable := FALSE,
//			bCurrentAlarmState := bDeviceCurrentAlarmState,
//			bCurrentWarningState := FALSE,
//			tAlarmDelay := tAlarmDelay_D,
//			bAlarm => bFaultAlarm,
//			bWarning => bFaultWarning
//			);
			
//		IF bFaultAlarm THEN
//			GVL_IO.aInterlock[1].0 := TRUE; //Alarm Trig
//			GVL_IO.nCaseSignalTower := 1; // Signal Tower RED - Alarm
//			//팝업 표시
//			wAlarm := ROR(GVL_IO.aInterlock[2], (i+13));
//			wAlarm.0 := TRUE;
//			GVL_IO.aInterlock[2] := ROL(wAlarm, (i+13));
//		END_IF
//	END_FOR
END_ACTION

ACTION _Button_Reset_Warning:
//IF GVL_IO.aInterlockEnable[1].0 THEN //알람 리셋 버턴을 눌렀을 때
//	GVL_IO.aInterlock[1].0 := FALSE; //Alarm Trig Reset
//	GVL_IO.aInterlockEnable[1].0 := FALSE; //버턴 초기화
//	GVL_IO.nCaseSignalTower := 4; // Signal Tower Blue - Idle
//END_IF
//IF GVL_IO.aInterlockEnable[1].1 THEN //주의 리셋 버턴을 눌렀을 때
//	GVL_IO.aInterlock[1].1 := FALSE; //Warmomg Trig Reset
//	GVL_IO.aInterlockEnable[1].1 := FALSE; //버턴 초기화
//	GVL_IO.nCaseSignalTower := 4; // Signal Tower Blue - Idle
//END_IF
END_ACTION

ACTION _DigitalInput:
bMaintKey := GVL_IO_REACTOR_CABINET.DI_01_MaintenanceModeKey;
bPowerResetSwitch := GVL_IO_GAS_CABINET.DI_01_ResetButton;
//jhkang Main Power Monitor 가 뭔가 ? 
//7. 순간정전 되었다가 전기가 다시 살아 났을 때,
// UPS는 전원이 살아있고, 히터, 펌프, bath는 전기가 나갔을 때 (아직 명확한 로직이 없음)

//jhkang_251112
//bMainPowerMonitor := GVL_IO.aDigitalInputIO[7].5; /// ??????? 이게 뭐지 ?
END_ACTION

END_PROGRAM

// ---- POUs/P17_DOROperation.TcPOU
PROGRAM P17_DOROperation
VAR
	bDOROn				: BOOL; //UI Input Button
	bDOROff				: BOOL; //UI Input Button
	fTresholdPressure	: REAL;
	fTresholdCount		: REAL;
	bPressureEnable 	: BOOL;
	bCountEnable		: BOOL;

	isDOROnState		: BOOL := FALSE; //DOR ON State
	bError				: INT; //0: No Err, 1: Vacuum Fail, 2: Vacuum Release, 3: Try out
	nWaitCounter		: INT;

	(* Input *)
	bVacSwitch			: BOOL; //Push Switch
	bAtmSwitch			: BOOL; //Push Switch
	(* Pressure Transducer *)
	nPressurePV			: INT;
	rPressurePV_Torr	: REAL;
	(* Output *)
	bVacLED				: BOOL;
	bAtmLED				: BOOL;
	bV_DORVac			: BOOL; //V34 Valve
	bV_DORFill			: BOOL; //V35 Valve
	
	(* DOR Condition Operation Parameter *)
	rTrigSwitch			: R_TRIG;
	TimerOnLED			: TON;
	TimerVacSwitch		: TON;
	TimerAtmSwitch		: TON;
	TimerWaitCheck		: TON;
	TimerVacRealease	: TON;
	nCase				: INT := 0;
	nTresholdCount		: INT;
	nTryCount			: INT;
	bVacuumRealse		: BOOL;
	//Temperatur Variable
	bTest				: BOOL;
	nTest				: INT;
END_VAR

VAR CONSTANT
	KL3464MaxValueP		: REAL := 16383; //1 ~ 5VDC, 0 ~ 100kPa(1bar), PG35
	SlopeFactor			: REAL := 0.007617887; //100kPa/(16383-3256)
END_VAR

////jhkang_251112
////인터락 재 확인
//// Double O-Ring Vacuum Condition
//_DigitalInput();
//_DOR_ON();
//_DOR_OFF();
//_VACUUM_RELEASE();

////알람 리셋
//IF GVL_IO.aInterlockEnable[1].0 OR GVL_IO.aInterlockEnable[1].1 THEN
//	bError := 0;
//END_IF

//_DigitalOutput();

ACTION _DigitalInput:
//jhkang_251112
//(* Read from Device Value *)
//// DOR Operation Switch
//bVacSwitch 			:= GVL_IO_REACTOR_CABINET.DI_01_DORVACButton; //Switch Input
//bAtmSwitch 			:= GVL_IO_REACTOR_CABINET.DI_01_DORATMButton; //Switch Input
//nPressurePV 		:= GVL_IO_REACTOR_CABINET.AI_07_S05_DORPressurePV;
//rPressurePV_Torr 	:= F_GetDorPressure(nPressurePV);

//fTresholdPressure 	:= GVL_IO.aInterlockSet[11]; // Dor Pressure Limit
//fTresholdCount 		:= GVL_IO.aInterlockSet[12]; // Dor Retry Count

//bPressureEnable 	:= GVL_IO.aInterlockEnable[1].5; // Dor Pressure Limit
//bCountEnable 		:= GVL_IO.aInterlockEnable[1].6; // Dor Retry Count
//nTresholdCount 		:= REAL_TO_INT(fTresholdCount); //Try One more Vacuum
END_ACTION

ACTION _DigitalOutput:
//jhkang_251112
//(* Write to Device Value *)
//// Cover Operation Switch Lamp

//GVL_INTERFACE_UI.aOutputSolValve.21:= bV_DORVac; //V34
//GVL_INTERFACE_UI.aOutputSolValve.22:= bV_DORFill; //V35
//GVL_IO.aInputState[4].10 :=bV_DORVac;

//GVL_IO_REACTOR_CABINET.DO_05_DORVACButtonLamp := bVacLED;
//GVL_IO_REACTOR_CABINET.DO_06_DORATMButtonLamp := bAtmLED;

//GVL_IO.nDorOperationError := bError;
////jhkang isDOROnState 뭐냐 
//GVL_IO.bDorState := isDOROnState;
END_ACTION

ACTION _DOR_OFF:
//jhkang_251112
//(* If Vacuum 'OFF' Switch Press, Change DOR Vent(Fill, Atm) State *)
////DOR Operation Signal generation
//TimerAtmSwitch(IN:=bAtmSwitch, PT:=T#100MS);
//rTrigSwitch(CLK:=TimerAtmSwitch.Q);

//IF rTrigSwitch.Q AND P90_Interlock.bDorOffEnable THEN
//	nCase := 2;
//END_IF

//CASE nCase OF
//	2:
//		(* Blink Switch LED *)
//		TimerOnLED(IN:=TRUE, PT:=T#500MS);
//		IF TimerOnLED.Q THEN
//			TimerOnLED(IN:=FALSE);
//			bAtmLED := NOT(bAtmLED);
//		END_IF
		
//		TimerWaitCheck(IN:=TRUE, PT:=T#10S);
//		nWaitCounter := TIME_TO_INT(TimerWaitCheck.ET/1000);
//		IF TimerWaitCheck.Q THEN
//			TimerWaitCheck(IN:=FALSE);
//			bVacLED			:= FALSE;
//			bV_DORVac 		:= FALSE; //V34 Close
//			bV_DORFill		:= TRUE; //V35 Open
//			nCase			:= 20;
//		END_IF
//	20:
//		TimerWaitCheck(IN:=TRUE, PT:=T#5S);
//		IF TimerWaitCheck.Q THEN
//			bVacLED			:= FALSE;
//			bV_DORFill		:= FALSE;
//			isDOROnState 	:= FALSE;
//			bAtmLED			:= TRUE;
//			nCase			:= 0;
//		END_IF
//END_CASE
END_ACTION

ACTION _DOR_ON:
//jhkang_251112
//(* If Vacuum 'ON' Switch Press, Change DOR Vacuum State *)
////DOR Operation Signal generation
////TimerVacSwitch(IN:=bVacSwitch OR bDOROn, PT:=T#100MS);
//TimerVacSwitch(IN:=bVacSwitch, PT:=T#100MS);
//rTrigSwitch(CLK:=TimerVacSwitch.Q);

//IF rTrigSwitch.Q AND GVL_IO.bDorOnEnable THEN
//	nCase 		:= 1;
//	nTryCount 	:= 1; //Try One more Vacuum 
//END_IF

//CASE nCase OF
//	1: //Initialize
//		isDOROnState := FALSE;
//		bV_DORVac 	:= TRUE; //V34 Open
//		bV_DORFill	:= FALSE; //V35 Close
//		bAtmLED		:= FALSE;
//		TimerWaitCheck(IN:=FALSE);	
//		nCase := 10;
		
//	10: //Wait and Vacuum Check
//		(* Blink Switch LED *)
//		TimerOnLED(IN:=TRUE, PT:=T#500MS);
//		IF TimerOnLED.Q THEN
//			TimerOnLED(IN:=FALSE);
//			bVacLED := NOT(bVacLED);
//		END_IF

//		TimerWaitCheck(IN:=TRUE, PT:=T#5S);
//		IF TimerWaitCheck.Q THEN
//			IF rPressurePV_Torr < fTresholdPressure THEN
//				bV_DORVac 		:= FALSE; //V34 Close
//				isDOROnState 	:= TRUE;
//				bVacLED 		:= TRUE; //Switch LED
//				bError			:= 0;
//				nCase 			:= 0;
//			ELSIF nTryCount < nTresholdCount THEN
//				TimerWaitCheck(IN:=FALSE);
//				nTryCount 		:= nTryCount + 1;				
//				nCase 			:= 1;
//			ELSE
//				bV_DORVac 		:= FALSE; //V34 Close
//				isDOROnState 	:= FALSE;
//				bVacLED			:= FALSE; //Switch LED
//				bError			:= 1; // Vacuum Fail
//				nCase			:= 0;
//			END_IF
//		END_IF
//END_CASE
END_ACTION

ACTION _VACUUM_RELEASE:
//jhkang_251112

//(* If Vacuum 'ON' State, Check the Vacuum range *)
//IF isDOROnState AND rPressurePV_Torr > fTresholdPressure AND nTryCount < 3 THEN
//	bError := 2; // Vacuum release
//	TimerVacRealease(IN:=TRUE, PT:=T#2S);
	
//	(* Blink Vac Switch LED *)
//	TimerOnLED(IN:=TRUE, PT:=T#500MS);
//	IF TimerOnLED.Q THEN
//		TimerOnLED(IN:=FALSE);
//		bVacLED := NOT(bVacLED);
//	END_IF

//	IF TimerVacRealease.Q  THEN
//		TimerVacRealease(IN:=FALSE);
//		nTryCount 		:= nTryCount + 1;
//		bV_DORVac 		:= FALSE;//Vacuum Valve OFF
//		bVacLED := TRUE;
//	ELSE
//		bV_DORVac 		:= TRUE;//Vacuum Valve ON
//	END_IF
	
//ELSIF bError = 2 THEN
//	bV_DORVac := FALSE;
//	bError := 0;
	
//ELSIF nTryCount >= 3 THEN
//	bV_DORVac := FALSE;
//	bError := 3; //Vacuum Released
//END_IF
END_ACTION

END_PROGRAM

// ---- POUs/P22_Background_ThermalBath.TcPOU
PROGRAM P22_Background_ThermalBath
VAR
	(* background communication with the KL6031 terminal (22byte)
	Thermal Bath(HEBC002-WA10) x 6EA *)
	fbCtrl		: SerialLineControl;
	bCtrlError	: BOOL;
	eCtrlErrorID	: ComError_t;
	fbConfig		: KL6configuration;
	bConfigError	: BOOL;
	eConfigErrorID: ComError_t;
	bConfigExe	: BOOL := TRUE;
	(* 	I/O variables for a KL6031 terminal*)

END_VAR

(*
The SerialLineControl function block is supposed to be called in every PLC cycle.
It communicates with the serial line hardware device and transmits or receives data.
The SerialLineControl can be called in the standard task (e.g.for PcCOM port usage) 
or in a separate fast task (e.g.for terminal usage) as well.
A fast separate task will be necessary at high baud rates or with KL6001 terminals 
which have a small process image (3 or 5 data bytes only)
TB: Thermal Bath x 6EA
Maker: SMC
Model: HEBC002-WA10
Temp Range: -15 ~60℃
RS485: 9600, DataBit(8), Parity(None), StopBit(1)
BCC Check : X
*)

fbCtrl(
	Mode:= SERIALLINEMODE_KL6_22B_STANDARD,
	pComIn:= ADR(GVL_Serial.stIn_KL6031_TB),
	pComOut:= ADR(GVL_Serial.stOut_KL6031_TB),
	SizeComIn:= SIZEOF(GVL_Serial.stIn_KL6031_TB),
	Error=> ,
	ErrorID=> ,
	TxBuffer:= GVL_Serial.TxBufferTB,
	RxBuffer:= GVL_Serial.RxBufferTB );
	
IF fbCtrl.Error THEN
	bCtrlError := TRUE;
	eCtrlErrorID := fbCtrl.ErrorID;
END_IF

END_PROGRAM

// ---- POUs/P50_RecipeControl.TcPOU
PROGRAM P50_RecipeControl
VAR
	nRcpIndex		: INT;
	eRecipeRun		: E_RecipeRun ; //레시피 상태
	fbAnalogDeviceRampControl : FB_AnalogDeviceRampControl;
	fbRecipeAnalogInputControlSequencer: FB_RecipeAnalogControlInputSequencer;
	fbValveControl: FB_ValveControl;
	
	Pause_TON		: TON;
	Ramp_TON		: FB_TON_Pausable;
	Hold_TON		: FB_TON_Pausable;
	
	loopCount		: ARRAY[1..100] OF INT;
	i				: INT;
END_VAR
VAR CONSTANT
	Pause_MAX		: TIME := T#1800S;
END_VAR

//jhkang_251112
//CASE GVL_INTERFACE_UI.recipe.control.cmd_RcpOperation OF
//	0: //Init State
// 		f_ResetTimersAndRCPTimes(fbPause_TON := Pause_TON, fbRamp_TON := Ramp_TON, fbHold_TON := Hold_TON);
		
//		FOR i:=1 TO GVL_INTERFACE_UI.recipe.iRcpTotalStep DO
//			loopCount[i] := GVL_INTERFACE_UI.recipe.aRecipe[i].iRecipe[5];
//		END_FOR
		
//		nRcpIndex := 0;
//		GVL_INTERFACE_UI.recipe.control.userState := 0;
//		eRecipeRun := E_RecipeRun.Initial;
//		GVL_IO.nCaseSignalTower := 5; // White - Idle

//	10: //RUN
//		IF nRcpIndex = 0 THEN
//			nRcpIndex := 1;
//		END_IF
//		fbAnalogDeviceRampControl();
						
//		// CASE 문을 이용한 상태 머신 구현
//		CASE eRecipeRun OF
//			E_RecipeRun.Initial:
//				f_ResetTimersAndRCPTimes(fbPause_TON := Pause_TON, fbRamp_TON := Ramp_TON, fbHold_TON := Hold_TON);
//				fbRecipeAnalogInputControlSequencer(rRecipe := GVL_INTERFACE_UI.recipe.aRecipe[nRcpIndex].rRecipe, rampTime:= TO_UINT(GVL_INTERFACE_UI.recipe.aRecipe[nRcpIndex].iRecipe[2]));
//				fbValveControl(valveSetting:= GVL_INTERFACE_UI.recipe.aRecipe[nRcpIndex].dRecipe);
//				GVL_INTERFACE_UI.recipe.control.userState := 10;// Recipe Running
//				GVL_IO.nCaseSignalTower := 3;
//				eRecipeRun := E_RecipeRun.Ramp;
				
//			E_RecipeRun.Ramp: // Ramp 수행
//				Ramp_TON(IN:=TRUE, PT:= GVL_INTERFACE_UI.recipe.aRecipe[nRcpIndex].iRecipe[2] * T#1S, ET=>GVL_INTERFACE_UI.recipe.control.RecipeRunET.ET);
//				GVL_INTERFACE_UI.recipe.control.RecipeRunET.Mode := E_RecipeRunETMode.Ramp;
//				IF Ramp_TON.Q THEN
//					Ramp_TON(IN:=FALSE);
//					eRecipeRun := E_RecipeRun.CheckHoldTemp;
//				END_IF				
				
//			E_RecipeRun.CheckHoldTemp: //Hold Temp 확인
//				IF GVL_INTERFACE_UI.recipe.aRecipe[nRcpIndex].cTemp = 0.0 THEN
//					Hold_TON(IN:=TRUE, PT:= GVL_INTERFACE_UI.recipe.aRecipe[nRcpIndex].iRecipe[3] * T#1S, ET=>GVL_INTERFACE_UI.recipe.control.RecipeRunET.ET);
//					GVL_INTERFACE_UI.recipe.control.RecipeRunET.Mode := E_RecipeRunETMode.Hold;
//					IF Hold_TON.Q THEN
//						Hold_TON(IN:=FALSE);
//						eRecipeRun := E_RecipeRun.End; // 레시피 첫 Column 실행
//					END_IF
//				ELSIF GVL_INTERFACE_UI.aAnalogController[E_aAnalogInputIO_Index.E_PV_Susceptor_Temp].pv < GVL_INTERFACE_UI.recipe.aRecipe[nRcpIndex].cTemp THEN //서셉터 온도가 Wait 온도보다 낮을 때
//					Hold_TON(IN:=FALSE);
//					eRecipeRun := E_RecipeRun.End; // 레시피 첫 Column 실행
//				ELSE // 서셉터 온도가 Wait 온도보다 높을 때
//					;// 떨어질 때까지 기다림
//				END_IF
				
//			E_RecipeRun.End: // 다음 Step 이동 (루프 마지막 단계일 경우, 다음 Step 이동 또는 루프 처음단계로 점프)
//				loopCount[nRcpIndex] := loopCount[nRcpIndex] - 1;
//				nRcpIndex := nRcpIndex + 1 - (GVL_INTERFACE_UI.recipe.aRecipe[nRcpIndex].iRecipe[4]) * MIN(loopCount[nRcpIndex], 1);
//				IF nRcpIndex > GVL_INTERFACE_UI.recipe.iRcpTotalStep THEN
//					GVL_INTERFACE_UI.recipe.control.cmd_RcpOperation := 50;
//				END_IF
//				eRecipeRun := E_RecipeRun.Initial;
//		END_CASE
		
//	20: //PAUSE
//		CASE eRecipeRun OF
//			E_RecipeRun.Ramp:
//				Ramp_TON(PAUSE:=TRUE);		
//			E_RecipeRun.CheckHoldTemp:
//				Hold_TON(PAUSE:=TRUE);
//		END_CASE
		
//		Pause_TON(IN:=TRUE, PT:= Pause_MAX, ET=>GVL_INTERFACE_UI.recipe.control.Pause_ET); //최대 홀드 시간이 지나면 다음 스텝으로 넘거감
//		IF Pause_TON.Q THEN
//			Pause_TON(IN:=FALSE);
//			eRecipeRun := E_RecipeRun.End; // 레시피 첫 Column 실행
//		END_IF

//		GVL_INTERFACE_UI.recipe.control.userState := 20;
//		GVL_IO.nCaseSignalTower := 5;
		
//	30: //RESTART
//		Pause_TON(IN:=FALSE);
//		CASE eRecipeRun OF
//			E_RecipeRun.Ramp:
//				Ramp_TON(PAUSE:=FALSE);
			
//			E_RecipeRun.CheckHoldTemp:
//				Hold_TON(PAUSE:=FALSE);
//		END_CASE

//		GVL_INTERFACE_UI.recipe.control.Pause_ET := T#0S;
//		GVL_INTERFACE_UI.recipe.control.userState := 10;
//		GVL_INTERFACE_UI.recipe.control.cmd_RcpOperation := 10;	
//		GVL_IO.nCaseSignalTower := 3;
		
//	40: //STOP
//		f_ResetTimersAndRCPTimes(fbPause_TON := Pause_TON, fbRamp_TON := Ramp_TON, fbHold_TON := Hold_TON);
//		F_StopAnalogRamping_ForRecipe();
//		GVL_INTERFACE_UI.recipe.control.userState := 40;
//		GVL_IO.nCaseSignalTower := 5;
		
//	50: //END
//		f_ResetTimersAndRCPTimes(fbPause_TON := Pause_TON, fbRamp_TON := Ramp_TON, fbHold_TON := Hold_TON);
//		GVL_INTERFACE_UI.recipe.control.userState := 50;
//		fbAnalogDeviceRampControl();
//		GVL_IO.nCaseSignalTower := 5;
		
//	60: //SKIP
//		IF E_RecipeRun.Ramp <= eRecipeRun  AND  eRecipeRun <= E_RecipeRun.CheckHoldTemp THEN
//			eRecipeRun := E_RecipeRun.End;
//		END_IF
//		GVL_INTERFACE_UI.recipe.control.cmd_RcpOperation := 10;
//		GVL_INTERFACE_UI.recipe.control.Pause_ET := T#0S;
//END_CASE
//GVL_INTERFACE_UI.recipe.control.iRcpStepN := nRcpIndex;

END_PROGRAM

// ---- POUs/FB_AnalogDeviceRampControl.TcPOU
FUNCTION_BLOCK FB_AnalogDeviceRampControl
VAR
	i : UINT;
END_VAR

FOR i:=1 TO GVL_CONSTANT.NumFlowController DO
	GVL_IO.io.analog.aAnalogOutputIO[i] := LREAL_TO_INT(GVL_INTERFACE_UI.aAnalogController[i].cvController.rControlValue); //Write to Device
	GVL_INTERFACE_UI.aAnalogController[i].cvController();
END_FOR


//Temp Controller

GVL_IO.ControlDevice.TEMP_CONTROLLER.SET_TEMP_SV := LREAL_TO_WORD(GVL_INTERFACE_UI.aAnalogController[E_aAnalogInputIO_Index.E_PV_Susceptor_Temp].cvController.rControlValue * 10 )  ; //Write to Temperature Controller
GVL_INTERFACE_UI.aAnalogController[E_aAnalogInputIO_Index.E_PV_Susceptor_Temp].cvController();

//Temp Pressure Controller				
GVL_IO.ControlDevice.THROTTLE_VALVE.SET_PRESSURE := LREAL_TO_WORD(GVL_INTERFACE_UI.aAnalogController[E_aAnalogInputIO_Index.E_PV_Reactor_Pressure].cvController.rControlValue); //Write to Pressure Controller
GVL_INTERFACE_UI.aAnalogController[E_aAnalogInputIO_Index.E_PV_Reactor_Pressure].cvController();

//jhkang_251112
//아래 항목 누락
//Rotation Controller		
//GVL_IO.ControlDevice.rRotation_ControlValue := LREAL_TO_REAL(GVL_INTERFACE_UI.aAnalogController[E_aAnalogInputIO_Index.E_PV_susceptorRotation].cvController.rControlValue); //Write to Rotation Controller (rpm)
//GVL_INTERFACE_UI.aAnalogController[E_aAnalogInputIO_Index.E_PV_susceptorRotation].cvController();

END_FUNCTION_BLOCK

// ---- POUs/FB_RecipeAnalogControlInputSequencer.TcPOU
FUNCTION_BLOCK FB_RecipeAnalogControlInputSequencer
VAR_INPUT
	rampTime: UINT;
END_VAR
VAR_IN_OUT
	rRecipe: ARRAY[1..(GVL_CONSTANT.NumAnalogController)] OF REAL;
END_VAR
VAR
	i: UINT;
END_VAR

FOR i := 1 TO GVL_CONSTANT.NumAnalogController DO
	GVL_INTERFACE_UI.aAnalogController[i].cvController.input.restart := TRUE;
	GVL_INTERFACE_UI.aAnalogController[i].cvController.input.rampTime := rampTime; 
	GVL_INTERFACE_UI.aAnalogController[i].cvController.input.targetValue := rRecipe[i];
END_FOR

END_FUNCTION_BLOCK

// ---- POUs/FB_ValveControl.TcPOU
FUNCTION_BLOCK FB_ValveControl
VAR_INPUT
	valveSetting: DWORD; 
END_VAR

//jhkang_251112
//(* Solenoid Valve Mapping *)
//GVL_INTERFACE_UI.aOutputSolValve.0 := valveSetting.0; //V01 B/G N2 In
//GVL_INTERFACE_UI.aOutputSolValve.1 := valveSetting.1;
//GVL_INTERFACE_UI.aOutputSolValve.2 := valveSetting.2;
//GVL_INTERFACE_UI.aOutputSolValve.3 := valveSetting.3;
//GVL_INTERFACE_UI.aOutputSolValve.4 := valveSetting.4;
//GVL_INTERFACE_UI.aOutputSolValve.5 := valveSetting.5;
//GVL_INTERFACE_UI.aOutputSolValve.6 := valveSetting.6;
//GVL_INTERFACE_UI.aOutputSolValve.7 := valveSetting.7;

//GVL_INTERFACE_UI.aOutputSolValve.8 := valveSetting.8;
//GVL_INTERFACE_UI.aOutputSolValve.9 := valveSetting.9;
//GVL_INTERFACE_UI.aOutputSolValve.10 := valveSetting.10;
//GVL_INTERFACE_UI.aOutputSolValve.11 := valveSetting.11;
//GVL_INTERFACE_UI.aOutputSolValve.12 := valveSetting.12;
//GVL_INTERFACE_UI.aOutputSolValve.13 := valveSetting.13;
//GVL_INTERFACE_UI.aOutputSolValve.14 := valveSetting.14;
//GVL_INTERFACE_UI.aOutputSolValve.15 := valveSetting.15;

//GVL_INTERFACE_UI.aOutputSolValve.16 := valveSetting.16; 
//GVL_INTERFACE_UI.aOutputSolValve.17 := valveSetting.17;
//GVL_INTERFACE_UI.aOutputSolValve.18 := valveSetting.18;
//GVL_INTERFACE_UI.aOutputSolValve.19 := valveSetting.19;
////GVL_INTERFACE_UI.aOutputSolValve.20 := valveSetting.20;

END_FUNCTION_BLOCK

// ---- POUs/P31_PriorityControl.TcPOU
PROGRAM P31_PriorityControl
VAR
	fbAnalogDeviceRampControl : FB_AnalogDeviceRampControl;
	pr_TON: TON;
END_VAR
VAR_OUTPUT
	complete : BOOL;
END_VAR

pr_TON(IN := TRUE, PT := (1 + GVL_INTERFACE_UI.aAnalogController[1].cvController.input.rampTime) * T#1S);
fbAnalogDeviceRampControl();
IF pr_TON.Q = TRUE THEN
	pr_TON(IN := FALSE);
	complete := TRUE;
ELSE 
	complete := FALSE;
END_IF

END_PROGRAM

// ---- POUs/P60_UpdatePV.TcPOU
PROGRAM P60_UpdatePV
VAR
	i: INT;
END_VAR

//jhkang_251112
//FOR i:=1 TO E_aAnalogInputIO_Index.E_PV_EPC_04 DO
//	GVL_INTERFACE_UI.aAnalogController[i].pv := INT_TO_REAL(GVL_IO.GVL_IO.io.analog.aAnalogInputIO[i]) / GVL_CONSTANT.EL3064MaxValueH * GVL_CONSTANT.AnalogControllerOutputVoltage;
//END_FOR

//GVL_INTERFACE_UI.aAnalogController[E_aAnalogInputIO_Index.E_PV_Susceptor_Temp].pv := WORD_TO_REAL(GVL_IO.wE3508_PV);
//GVL_INTERFACE_UI.aAnalogController[E_aAnalogInputIO_Index.E_PV_Reactor_Pressure].pv := WORD_TO_REAL(GVL_IO.wIqPlus_CDG2_PV);
//GVL_INTERFACE_UI.aAnalogController[E_aAnalogInputIO_Index.E_PV_susceptorRotation].pv := GVL_IO.nRotation_Converted_PV;

END_PROGRAM

// ---- POUs/P91_Monitoring.TcPOU
PROGRAM P91_Monitoring
VAR
	TimeCycle			: TON;
	i 					: INT;
	idx					: INT;
	
	(*Utility Input*)
	bUtilityFault		: BYTE;	
	JhValue_DOR: REAL;
	JhValue_EXHAUST: REAL;
END_VAR

//jhkang

(* Read from Utility Device*)

//jhkang butilityFault 는 어떤 것인가?
bUtilityFault.0		:= GVL_IO_GAS_CABINET.DI_05_ExternalH2GasCabinetFault;
bUtilityFault.1		:= GVL_IO_GAS_CABINET.DI_05_ExternalH2SGasCabinetFault;
bUtilityFault.2		:= GVL_IO_GAS_CABINET.DI_05_ExternalH2SeGasCabinetFault;
bUtilityFault.3		:= GVL_IO_GAS_CABINET.DI_05_ExternalUserInputAlarm;

TimeCycle(IN:=TRUE, PT:=T#100MS); // 100MS Refresh Reading Time
IF TimeCycle.Q THEN
	TimeCycle(IN:=FALSE);
	_DOR_EXHAUST()
;

	// Reactor Ultimate Pressure Gauge
	GVL_INTERFACE_UI.aMonitoring_PV[1] := GVL_IO.io.analog.aAnalogInputIO[E_aAnalogInputIO_Index.E_PV_Ultimate_Pressure] / GVL_CONSTANT.EL3064MaxValue * 10; //Ultimate Pressure 10Torr, 0~10V, Cal. x10
	GVL_INTERFACE_UI.aMonitoring_PV[2] := JhValue_EXHAUST;
	GVL_INTERFACE_UI.aMonitoring_PV[3] := JhValue_DOR;
	GVL_INTERFACE_UI.aMonitoring_PV[4] := GVL_IO.io.analog.aAnalogInputIO[E_aAnalogInputIO_Index.E_PV_GAS_Pressure_N2] / GVL_CONSTANT.EL3064MaxValue * 10; //N2 Cal. 6.89 bar  
	GVL_INTERFACE_UI.aMonitoring_PV[5] := GVL_IO.io.analog.aAnalogInputIO[E_aAnalogInputIO_Index.E_PV_GAS_Pressure_H2] / GVL_CONSTANT.EL3064MaxValue * 10; //H2 Cal. 6.89 bar
	GVL_INTERFACE_UI.aMonitoring_PV[6] := GVL_IO.io.analog.aAnalogInputIO[E_aAnalogInputIO_Index.E_PV_GAS_Pressure_H2S] / GVL_CONSTANT.EL3064MaxValue * 10; //NH3 Cal. 6.89 bar
	GVL_INTERFACE_UI.aMonitoring_PV[7] := GVL_IO.io.analog.aAnalogInputIO[E_aAnalogInputIO_Index.E_PV_GAS_Pressure_H2Se] / GVL_CONSTANT.EL3064MaxValue * 10; // Cal. 6.89 bar
	GVL_INTERFACE_UI.aMonitoring_PV[8] := GVL_IO.io.analog.aAnalogInputIO[E_aAnalogInputIO_Index.E_PV_CoolingWafer_SH] * 0.1; //  // PT100, Shower Head, Cal. 0.1
//	GVL_INTERFACE_UI.aMonitoring_PV[9] := GVL_IO.io.analog.aAnalogInputIO2[1] / GVL_CONSTANT.EL3102MAxValue * 10;
//	GVL_INTERFACE_UI.aMonitoring_PV[10] := GVL_IO.io.analog.aAnalogInputIO2[2] / GVL_CONSTANT.EL3102MAxValue * 10 ; 
	GVL_INTERFACE_UI.aMonitoring_PV[11] := WORD_TO_REAL(P11_E3508.wE3508_PowerRate)*0.1; //divided to 10 PowerRate
	GVL_INTERFACE_UI.aMonitoring_PV[12] := P12_IQ_PLUS.wByteValvePosition_PV_Monitoring;
	GVL_INTERFACE_UI.aMonitoring_PV[13] := P14_ThermalBath.rTemperature_PV[1];
	GVL_INTERFACE_UI.aMonitoring_PV[14] := P14_ThermalBath.rTemperature_PV[2];
	GVL_INTERFACE_UI.aMonitoring_PV[15] := P14_ThermalBath.rTemperature_PV[3];
	GVL_INTERFACE_UI.aMonitoring_PV[16] := P14_ThermalBath.rTemperature_PV[4];
	
//jhkang_251112
//aController_PV 협의 필요 
//	GVL_INTERFACE_UI.aMonitoring_PV[17] := GVL_IO.aController_PV[E_aAnalogInputIO_Index.E_PV_MFC_01];
	
//	IF  GVL_IO_VALVE.DO_00_V17GasH2SeManifoldRun = TRUE THEN
//		GVL_INTERFACE_UI.aMonitoring_PV[17]:=GVL_INTERFACE_UI.aMonitoring_PV[17] + GVL_IO.aController_PV[E_aAnalogInputIO_Index.E_PV_MFC_03];
//	END_IF
//		IF  GVL_IO_VALVE.DO_00_V18GasH2SManifoldRun = TRUE THEN
//		GVL_INTERFACE_UI.aMonitoring_PV[17]:=GVL_INTERFACE_UI.aMonitoring_PV[17] + GVL_IO.aController_PV[E_aAnalogInputIO_Index.E_PV_MFC_04];
//	END_IF
//		IF  GVL_IO_VALVE.DO_00_V19Source_4ChalcogenManifoldRun = TRUE THEN
//		GVL_INTERFACE_UI.aMonitoring_PV[17]:=GVL_INTERFACE_UI.aMonitoring_PV[17] + GVL_IO.aController_PV[E_aAnalogInputIO_Index.E_PV_MFC_08];
//	END_IF
	
	
	
//	GVL_INTERFACE_UI.aMonitoring_PV[18] := GVL_IO.aController_PV[E_aAnalogInputIO_Index.E_PV_MFC_02];
//	IF  GVL_IO_VALVE.DO_00_V14Source_1TMInManifoldRun = TRUE THEN
//		GVL_INTERFACE_UI.aMonitoring_PV[18]:=GVL_INTERFACE_UI.aMonitoring_PV[18] + GVL_IO.aController_PV[E_aAnalogInputIO_Index.E_PV_MFC_05];
//	END_IF
//	IF  GVL_IO_VALVE.DO_00_V15Source_2TMGaManifoldRun = TRUE THEN
//		GVL_INTERFACE_UI.aMonitoring_PV[18]:=GVL_INTERFACE_UI.aMonitoring_PV[18] + GVL_IO.aController_PV[E_aAnalogInputIO_Index.E_PV_MFC_06];
//	END_IF
//	IF  GVL_IO_VALVE.DO_00_V16Source_3DMSeManifoldRun = TRUE THEN
//		GVL_INTERFACE_UI.aMonitoring_PV[18]:=GVL_INTERFACE_UI.aMonitoring_PV[18] + GVL_IO.aController_PV[E_aAnalogInputIO_Index.E_PV_MFC_07];
//	END_IF
END_IF

ACTION _DOR_EXHAUST:
GVL_SEQUENCE.FB_DOR_PRESSURE_AVG(newValue:=F_GetDorPressure(GVL_IO.io.analog.aAnalogInputIO[E_aAnalogInputIO_Index.E_PV_DOR_PRESSURE]),Output=>JhValue_DOR);
GVL_SEQUENCE.FB_EXHAUST_AVG(newValue:=F_GetDorPressure(GVL_IO.io.analog.aAnalogInputIO[E_aAnalogInputIO_Index.E_PV_Exhaust_Pressure]),Output=>JhValue_EXHAUST);
END_ACTION

END_PROGRAM

// ---- FUNCTION/F_GetDorPressure.TcPOU
FUNCTION F_GetDorPressure : real
VAR_INPUT
	nPressurePV:INT;
END_VAR

VAR
	Value:REAL;
END_VAR

Value:= (10.0 / 32767.0) * nPressurePV;
F_GetDorPressure := (190* (Value) ) - 190;

END_FUNCTION

// ---- POUs/P92_Maintenance.TcPOU
PROGRAM P92_Maintenance
VAR
	(* Input *)
	//Light
	rTrigReactorCabinetSwitch	: R_TRIG;
	rTrigReactorCabinetMagnet 	: R_TRIG;
	fTrigReactorCabinetMagnet 	: F_TRIG;
	rTrigGasCabinetSwitch		: R_TRIG;
	rTrigGasCabinetMagnet		: R_TRIG;
	fTrigGasCabinetMagnet		: F_TRIG;

	bReactorCabinetLampSwitch : BOOL;
	bGasCabinetLampSwitch	: BOOL;
	
	bReactorCabientMagnet	: BOOL;
	bGasCabinetMagnet		: BOOL;
	bPowerDistributeMagnet	: BOOL;
	
	(* Output to Device *)
	// Cabinet Lamp
	bReactorCabinetLamp		: BOOL;
	bGasCabinetLamp			: BOOL;
	bPowerDistributeLamp	: BOOL;
	
	bSMPS24V480WFault		: BOOL;
	bSMPS24V72WFault		: BOOL;
	bSMPS15VPlusFault		: BOOL;
	bSMPS15VMinusFault		: BOOL;
	// Signal Tower
	bSignalTower			: BYTE;
	TimerSignalTower		: TON;
	bBuzzer					: BOOL;
	rTrigReactorDoorClose: R_TRIG;
END_VAR

(* Read from Device Value *)

// Reactor Cabinet Lamp
rTrigReactorCabinetSwitch(CLK:=GVL_IO_REACTOR_CABINET.DI_01_ReactorCabinetLampButton);
fTrigReactorCabinetMagnet(CLK:=GVL_IO_REACTOR_CABINET.DI_03_ReactorCabinetDoorClose);

IF rTrigReactorCabinetSwitch.Q OR rTrigReactorCabinetMagnet.Q OR fTrigReactorCabinetMagnet.Q THEN
	bReactorCabinetLamp := NOT(bReactorCabinetLamp);
END_IF

rTrigReactorDoorClose(CLK:=GVL_IO_REACTOR_CABINET.DI_03_ReactorCabinetDoorClose);
IF rTrigReactorDoorClose.Q THEN
	bReactorCabinetLamp:=FALSE;
END_IF


// Gas Delivery Cabinet Lamp
rTrigGasCabinetSwitch(CLK:= GVL_IO_GAS_CABINET.DI_01_GasCabinetLampButton);
rTrigGasCabinetMagnet(CLK:= GVL_IO_GAS_CABINET.DI_01_GasCabinetDoorClose);

IF rTrigGasCabinetSwitch.Q THEN
	bGasCabinetLamp := NOT(bGasCabinetLamp);
ELSIF fTrigGasCabinetMagnet.Q THEN
	bGasCabinetLamp := TRUE;
ELSIF rTrigGasCabinetMagnet.Q THEN
	bGasCabinetLamp := FALSE;
END_IF

IF GVL_IO_GAS_CABINET.DI_01_ControlCabinetDoorClose = TRUE THEN
	IF bPowerDistributeLamp THEN 
		bPowerDistributeLamp:=FALSE;
	END_IF
ELSE
	bPowerDistributeLamp := NOT(bPowerDistributeMagnet); //Magnet Switch	
END_IF
// Power Distribute Unit Lamp


_Action_Buzzer();
_Action_SignalTower();

(* Write to Device Value *)
GVL_IO_REACTOR_CABINET.DO_06_ReactorCabinetLamp := bReactorCabinetLamp;
GVL_IO_GAS_CABINET.DO_07_GasCabinetLamp := bGasCabinetLamp;
GVL_IO_GAS_CABINET.DO_07_ControlCabinetLamp := bPowerDistributeLamp;

ACTION _Action_Buzzer:
//jhkang_251112
//(* Buzzer On/Off *)
//IF bBuzzer <> GVL_IO.aInterlockEnable[1].2 THEN
//	bBuzzer := GVL_IO.aInterlockEnable[1].2;
//END_IF
END_ACTION

ACTION _Action_SignalTower:
//jhkang_251112

//(* Blink Signal Tower *)
//CASE GVL_IO.nCaseSignalTower OF
//	1: //RED 
//		TimerSignalTower(IN:=TRUE, PT:=T#500MS);
//		IF TimerSignalTower.Q THEN
//			TimerSignalTower(IN:=FALSE);
//			IF bSignalTower = 0 THEN
//				bSignalTower := 2#0000_0001; // RED
//			ELSE
//				bSignalTower := 0;
//			END_IF
//		END_IF

//	2: //YELLOW 
//		TimerSignalTower(IN:=TRUE, PT:=T#1S);
//		IF TimerSignalTower.Q THEN
//			TimerSignalTower(IN:=FALSE);
//			IF bSignalTower = 0 THEN
//				bSignalTower := 2#0000_0010; // YELLOW
//			ELSE
//				bSignalTower := 0;
//			END_IF
//		END_IF
//	3: //GREEN
//		TimerSignalTower(IN:=TRUE, PT:=T#1S);
//		IF TimerSignalTower.Q THEN
//			TimerSignalTower(IN:=FALSE);
//			IF bSignalTower = 0 THEN
//				bSignalTower := 2#0000_0100; // GREEN
//			ELSE
//				bSignalTower := 0;
//			END_IF
//		END_IF
//	4: //BLUE
//		bSignalTower := 2#0000_1000;
//	5: //WHITE
//		bSignalTower := 2#0001_0000;
//END_CASE

//GVL_IO_REACTOR_CABINET.DO_04_SignalTowerRed:=bSignalTower.0; //0:RED-Alarm,
//GVL_IO_REACTOR_CABINET.DO_04_SignalTowerOrange:=bSignalTower.1; //1:YELLOW,-Warning
//GVL_IO_REACTOR_CABINET.DO_04_SignalTowerGreen:=bSignalTower.2; //2:GREEN-Running
//GVL_IO_REACTOR_CABINET.DO_04_SignalTowerBlue:=bSignalTower.3; //3:BLUE-Idle
//GVL_IO_REACTOR_CABINET.DO_04_SignalTowerWhite:=bSignalTower.4; //4:WHITE-Maint
//GVL_IO_REACTOR_CABINET.DO_04_SignalTowerBuzzer:=bBuzzer; //5:BUZZER-Alarm
END_ACTION

END_PROGRAM

// ---- DEVICE/LINE HEATER/FB_TEMP_RAMPING.TcPOU
FUNCTION_BLOCK FB_TEMP_RAMPING
VAR_INPUT
	bExecute:BOOL;
	StartTemp:REAL;
	RampingTargetTemp:REAL;
	RampingTime:REAL;
END_VAR
VAR_OUTPUT
	OutputSetTemp:INT;
	bTempChangeFlag:BOOL;
	bBusy: BOOL;
END_VAR
VAR
	RingEdge: R_TRIG;
	fallEdge: F_TRIG;
	StartTemp_Bak:REAL;
	RampingTargetTemp_Bak:REAL;
	RampingTime_Bak:REAL;
	SeqStep: INT;
	nCycleCountms: INT;
	nCycleCountSec: INT;
	RampingTempPerSec:REAL;

	nDelayCount: INT;
END_VAR

RingEdge(CLK:=bExecute);
fallEdge(CLK:=bExecute);

IF RingEdge.Q THEN
	(*Ramping Start*)
	StartTemp_Bak:=StartTemp;
	RampingTargetTemp_Bak  := RampingTargetTemp;
	RampingTime_Bak := RampingTime;
	bBusy := TRUE;
	SeqStep:=10;
END_IF

IF fallEdge.Q THEN
	SeqStep:=0;
	bBusy := FALSE;
	bTempChangeFlag:=FALSE;
END_IF


CASE SeqStep OF
	0:(*IDE*)
		nCycleCountms:=0;
		nCycleCountSec:=0;
		nDelayCount:=0;

	10:(*Ramping Start*)
		IF RampingTime_Bak <=0 THEN
			RampingTime_Bak:=1;
		END_IF
		
		RampingTempPerSec := (RampingTargetTemp_Bak - StartTemp_Bak) / RampingTime_Bak;
		SeqStep:= 20;
		
	20:
		nCycleCountms :=  nCycleCountms+1;
		IF nCycleCountSec >= RampingTime_Bak THEN
			OutputSetTemp:=REAL_TO_INT(RampingTargetTemp_Bak);
			SeqStep:= 100;
		END_IF
		
		IF nCycleCountms >= 200 THEN
			nCycleCountms:=0;
			nCycleCountSec := nCycleCountSec+2;
			
			OutputSetTemp:= REAL_TO_INT(StartTemp + REAL_TO_INT( RampingTempPerSec * nCycleCountSec));
			
			IF RampingTime_Bak <= 1 THEN
				OutputSetTemp:=REAL_TO_INT(RampingTargetTemp_Bak);
			END_IF
			
			bTempChangeFlag:=TRUE;
		END_IF
		
		IF bTempChangeFlag = TRUE AND nCycleCountms >10 THEN
			bTempChangeFlag:=FALSE;
		END_IF
		
		
		
	100:
		nDelayCount:=nDelayCount+1;
		IF nDelayCount > 100 THEN
			bExecute:=FALSE;	
			SeqStep:=0;			
		END_IF

	
END_CASE

END_FUNCTION_BLOCK

// ---- DEVICE/LINE HEATER/FUNCTION/F_Temp_Write_Value.TcPOU
FUNCTION F_Temp_Write_Value : ST_Modbus_Send_Frame
VAR_INPUT
	Module_Number	:BYTE;
	Command_Index	:WORD;
	Write_Value		:WORD;
END_VAR
VAR
END_VAR

F_Temp_Write_Value.UnitID	:= Module_Number;
F_Temp_Write_Value.StartAddress	:= Command_Index;
F_Temp_Write_Value.sendQuantity	:= 1;
F_Temp_Write_Value.SendData[0]	:= Write_Value;

END_FUNCTION

// ---- FUNCTION/BOOL_TO_STRING_LHeaterON.TcPOU
FUNCTION BOOL_TO_STRING_LHeaterON : STRING
VAR_INPUT
	nHeaterNumber	: INT;
	bON				: BOOL;
END_VAR
VAR
	sString			: STRING;
	sHeaterNumber	: STRING;
END_VAR

////LH: Line Heater x 8EA -> 8Channel TIC 1EA
////Model: HANYOUNG NUX, MC9-8RD0SS32

////STRING : '$0201DWR,02,0302(CH_NO),0001(CH_1),0501(AT),0001(AT-ON)
//sString := '$0201DWR,02,0302,,0501,000$0D$0A';

////Convert to Channel from Heater Number
//sHeaterNumber := DINT_TO_DECSTR(nHeaterNumber, 4);
//sString := INSERT(sString,sHeaterNumber,15);

//IF bON = TRUE THEN
//	sString := INSERT(sString,'1',28);
//ELSE
//	sString := INSERT(sString,'0',28);
//END_IF

//BOOL_TO_STRING_LHeaterON := sString;

END_FUNCTION

// ---- FUNCTION/F_ReactorIndexToAnalogControllerIndex.TcPOU
FUNCTION F_ReactorIndexToAnalogControllerIndex : UINT
VAR_INPUT
	i : UINT;
END_VAR
VAR
END_VAR

F_ReactorIndexToAnalogControllerIndex := i + GVL_CONSTANT.NumFlowController;

END_FUNCTION

// ---- FUNCTION/Real_To_String_LineHeater.TcPOU
FUNCTION Real_To_String_LineHeater : STRING
VAR_INPUT
	rTemperatureSV 		: REAL;
	nHeaterNumber		: INT;
END_VAR
VAR
	wTemperature		: WORD;
	hStrTemp			: STRING;
	sHeaterNumber		: STRING;
	sString				: STRING;
	sSendString			: STRING;
END_VAR

////LH: Line Heater x 8EA -> 8Channel TIC 1EA
////Model: HANYOUNG NUX, MC9-8RD0SS32

//// Multiple decimal place point
//// STRING : '$0201DWR,03,0301(ZONE_NO),0001(ZONE_1),0302(CH_NO),0001(CH_1,sHeaterNumber),0401(SV), hStrTemp, $0D$0A'
//sString := '$0201DWR,03,0301,0001,0302,,0401,,$0D$0A';

////Convert to Channel from Heater Number
//sHeaterNumber := DINT_TO_DECSTR(nHeaterNumber, 4);
//sString := INSERT(sString,sHeaterNumber,25);
	
////Convert to String Type
//wTemperature := REAL_TO_WORD(rTemperatureSV);
//hStrTemp := WORD_TO_HEXSTR(wTemperature, 4, FALSE);
//Real_To_String_LineHeater := INSERT(sString,hStrTemp,35);

END_FUNCTION

// ---- FUNCTION/USINT_TO_WORD_jh.TcPOU
//2-USINT combine to 1-WORD converting using a bit operation
FUNCTION USINT_TO_WORD_jh : WORD
VAR_INPUT
	aInput: ARRAY[0..1]OF USINT; //Lower
END_VAR
VAR
	nWord_L : WORD; //Lower
	nWord_U : WORD; //Upper
END_VAR

USINT_TO_WORD_jh := TO_WORD(aInput[0]) OR SHL(TO_WORD(aInput[1]), 8);

END_FUNCTION

// ---- POUs/FB_OverLimitCheck.TcPOU
//*********************************************************************
// Function Block: FB_OverLimitCheck
// Description: 각 디바이스의 범위 초과 알람을 처리합니다.
// bEnable이 TRUE일 때만 알람 로직이 활성화됩니다.
//*********************************************************************
FUNCTION_BLOCK FB_OverLimitCheck
VAR_INPUT
	bAlarmEnable	: BOOL; //디바이스 활성화/비활성화 (TRUE = 활성화)
	bWarningEnable	: BOOL;
	fCurrentValue 	: REAL; //현재값
	fAlarmTreshold	: REAL; //알람 허용 임계값
	fWarningTreshold : REAL; //경고 허용 임계값
	tAlarmDelay		: TIME; //지연 시간
END_VAR
VAR_OUTPUT
	bAlarm			: BOOL; //허용 값 초과 경고 발생
	bWarning		: BOOL; //허용 값 초과 주의 발생
END_VAR
VAR
	//내부 변수 (인스턴스별로 독립적)
	fbAlarmTimer 		: TON;
	fbWarningTimer 	: TON;
 	bAlarmCondition 	: BOOL;
	bWarningCondition 	: BOOL; 
END_VAR

// bAlarmEnable이 TRUE일 때만 알람 로직 실행
IF bAlarmEnable THEN
	//허용값 알람 로직(지연 시간 적용)
	IF fCurrentValue > fAlarmTreshold THEN
		bAlarmCondition := TRUE;
	ELSE
		bAlarmCondition := FALSE;
	END_IF
	fbAlarmTimer(IN:=bAlarmCondition, PT:=tAlarmDelay);
	bAlarm := fbAlarmTimer.Q;
ELSE
	// bEnable이 FALSE일 경우, 모든 알람 및 타이머를 비활성화/리셋
    // Q 출력을 FALSE로 강제하고, IN 입력을 FALSE로 설정하여 타이머를 리셋합니다.
	bAlarm := FALSE;
	fbAlarmTimer(IN := FALSE, PT := tAlarmDelay); // 타이머 리셋
	bAlarmCondition := FALSE; // 조건 플래그도 리셋
END_IF

// bWarningEnable이 TRUE일 때만 알람 로직 실행
IF bWarningEnable THEN
	//허용값 주의 로직(지연 시간 적용)
	IF (fCurrentValue > fWarningTreshold) AND (fCurrentValue <= fAlarmTreshold ) THEN
		bWarningCondition := TRUE;
	ELSE
		bWarningCondition := FALSE;
	END_IF
	fbWarningTimer(IN:=bWarningCondition, PT:=tAlarmDelay);
	bWarning := fbWarningTimer.Q;
ELSE
	// bEnable이 FALSE일 경우, 모든 알람 및 타이머를 비활성화/리셋
    // Q 출력을 FALSE로 강제하고, IN 입력을 FALSE로 설정하여 타이머를 리셋합니다.
	bWarning := FALSE;
	fbWarningTimer(IN := FALSE, PT := tAlarmDelay); // 타이머 리셋
	bWarningCondition := FALSE; // 조건 플래그도 리셋
END_IF

END_FUNCTION_BLOCK

// ---- POUs/F_StopAnalogRamping_ForRecipe.TcPOU
FUNCTION F_StopAnalogRamping_ForRecipe
VAR
	i: UINT;
END_VAR

FOR i := 1 TO GVL_CONSTANT.NumAnalogController DO
	GVL_INTERFACE_UI.aAnalogController[i].cvController.input.restart := TRUE;
	GVL_INTERFACE_UI.aAnalogController[i].cvController.input.rampTime := 1; 
	GVL_INTERFACE_UI.aAnalogController[i].cvController.input.targetValue := LREAL_TO_REAL(GVL_INTERFACE_UI.aAnalogController[i].cvController.rControlValue);
END_FOR

END_FUNCTION

// ---- POUs/FUNCTION/FB_RINGBUFFER.TcPOU
FUNCTION_BLOCK FB_RINGBUFFER
VAR_INPUT
    newValue  : REAL;                  
END_VAR
VAR_OUTPUT
	Output: INT;
END_VAR
VAR
	bFirstStart:BOOL:=FALSE;
	arrValues : ARRAY[0..60] OF REAL;  
    sum: REAL := 0;          
   	SamplingCount:INT;        
	i: INT;
END_VAR

IF bFirstStart = FALSE THEN
	bFirstStart:=TRUE;
	
END_IF

SamplingCount:=60;


FOR i := SamplingCount TO 2 BY -1 DO
    arrValues[i] := arrValues[i-1];
END_FOR;

arrValues[1] := newValue;


sum := 0;
FOR i := 1 TO SamplingCount DO
    sum := sum + arrValues[i];
END_FOR;

Output := REAL_TO_INT(sum / SamplingCount);

END_FUNCTION_BLOCK

// ---- POUs/FUNCTION/F_StateValve_Process_Source.TcPOU
FUNCTION F_StateValve_Process_Source : bool
VAR_INPUT
END_VAR
VAR
END_VAR

F_StateValve_Process_Source:= GVL_IO_VALVE.DO_00_V01ChalcogenCarrierChange = FALSE AND
				GVL_IO_VALVE.DO_00_V02MOCarreirChange = FALSE  AND
				GVL_IO_VALVE.DO_00_V03H2SeSourceChange = FALSE  AND
				GVL_IO_VALVE.DO_00_V04H2SSourceChange = FALSE  AND
				GVL_IO_VALVE.DO_00_V05Source_1TMInCarrierChange = FALSE  AND
				GVL_IO_VALVE.DO_00_V06Source_1TMInBypass = FALSE  AND
				GVL_IO_VALVE.DO_00_V07Source_2TMGaCarrierChange = FALSE  AND
				GVL_IO_VALVE.DO_00_V08Source_2TMGaBypass = FALSE  AND
				GVL_IO_VALVE.DO_00_V09Source_3DMSeCarrierChange = FALSE  AND
				GVL_IO_VALVE.DO_00_V10Source_3DMSeBypass = FALSE  AND
				GVL_IO_VALVE.DO_00_V11Source_4ChalcogenCarrierChange = FALSE  and
				GVL_IO_VALVE.DO_00_V12Source_4ChalcogenBypass = FALSE;

END_FUNCTION

// ---- POUs/FUNCTION/F_StateValve_Process.TcPOU
FUNCTION F_StateValve_Process : bool
VAR_INPUT
END_VAR
VAR
END_VAR

F_StateValve_Process:= GVL_IO_VALVE.DO_00_V01ChalcogenCarrierChange = FALSE AND
				GVL_IO_VALVE.DO_00_V02MOCarreirChange = FALSE  AND
				GVL_IO_VALVE.DO_00_V03H2SeSourceChange = FALSE  AND
				GVL_IO_VALVE.DO_00_V04H2SSourceChange = FALSE ;

END_FUNCTION
